(********************* G.D S.p.A. - Technical Department ***********************************
This program has been generated automatically from Application Designer DE&F
********************************************************************************************)
PROGRAM dbg_csp_case_transport_os_minorplow
VAR
  bwd_di_shd : digital_input_shadow;
  fwd_di_shd : digital_input_shadow;
  shift_do_shd : digital_output_shadow;
  shift_sact_shd : digital_actuator_shadow;
END_VAR

_objects_manager();

IF	g_application_status <> APPLICATION_STATUS_RUNNING
THEN
	RETURN;
END_IF

CASE process_get_mode(CONVERSION_this := dbg_root.prc) OF
	MODE_ABSENT,
	MODE_INACTIVE:
		RETURN;
	MODE_TEST:
		RETURN;
END_CASE

ACTION _objects_manager:
IF	objects_initialization()
THEN
	digital_input_shadow_init(
		sim_mode:= SHADOW_SIMULATION_MODE_AUTOMATIC, 
		father:= csp_case_transport_os_minorplow.bwd_di, 
		process:= dbg_root.prc, 
		CONVERSION_this:= bwd_di_shd);

	digital_input_shadow_init(
		sim_mode:= SHADOW_SIMULATION_MODE_AUTOMATIC, 
		father:= csp_case_transport_os_minorplow.fwd_di, 
		process:= dbg_root.prc, 
		CONVERSION_this:= fwd_di_shd);

	digital_output_shadow_init(
		sim_mode:= SHADOW_SIMULATION_MODE_AUTOMATIC, 
		father:= csp_case_transport_os_minorplow.shift_do, 
		process:= dbg_root.prc, 
		CONVERSION_this:= shift_do_shd);

	digital_actuator_shadow_init(
		sim_mode:= SHADOW_SIMULATION_MODE_AUTOMATIC, 
		father:= csp_case_transport_os_minorplow.shift_sact, 
		process:= dbg_root.prc, 
		CONVERSION_this:= shift_sact_shd);

	RETURN;
END_IF

IF	objects_running()
THEN
	digital_input_shadow_cycle(bwd_di_shd);
	digital_input_shadow_cycle(fwd_di_shd);
	digital_output_shadow_cycle(shift_do_shd);
	digital_actuator_shadow_cycle(shift_sact_shd);
END_IF
END_ACTION

END_PROGRAM

// ---- _Debug/dbg_csp_case_transport_os_trailing.TcPOU

(********************* G.D S.p.A. - Technical Department ***********************************
This program has been generated automatically from Application Designer DE&F
********************************************************************************************)
PROGRAM dbg_csp_case_transport_os_trailing
VAR
  axis_shd : axis_shadow;
END_VAR

_objects_manager();

IF	g_application_status <> APPLICATION_STATUS_RUNNING
THEN
	RETURN;
END_IF

CASE process_get_mode(CONVERSION_this := dbg_root.prc) OF
	MODE_ABSENT,
	MODE_INACTIVE:
		RETURN;
	MODE_TEST:
		RETURN;
END_CASE

ACTION _objects_manager:
IF	objects_initialization()
THEN
	axis_shadow_init(
		sim_mode:= SHADOW_SIMULATION_MODE_AUTOMATIC, 
		father:= csp_case_transport_os_trailing.axis, 
		process:= dbg_root.prc, 
		CONVERSION_this:= axis_shd);

	RETURN;
END_IF

IF	objects_running()
THEN
	axis_shadow_cycle(axis_shd);
END_IF
END_ACTION

END_PROGRAM

// ---- _Debug/dbg_csp_case_transport_tensioner.TcPOU

(********************* G.D S.p.A. - Technical Department ***********************************
This program has been generated automatically from Application Designer DE&F
********************************************************************************************)
PROGRAM dbg_csp_case_transport_tensioner
VAR
  chain_tensioner_do_shd : digital_output_shadow;
  chain_tensioner_sact_shd : digital_actuator_shadow;
END_VAR

_objects_manager();

IF	g_application_status <> APPLICATION_STATUS_RUNNING
THEN
	RETURN;
END_IF

CASE process_get_mode(CONVERSION_this := dbg_root.prc) OF
	MODE_ABSENT,
	MODE_INACTIVE:
		RETURN;
	MODE_TEST:
		RETURN;
END_CASE

ACTION _objects_manager:
IF	objects_initialization()
THEN
	digital_output_shadow_init(
		sim_mode:= SHADOW_SIMULATION_MODE_AUTOMATIC, 
		father:= csp_case_transport_tensioner.chain_tensioner_do, 
		process:= dbg_root.prc, 
		CONVERSION_this:= chain_tensioner_do_shd);

	digital_actuator_shadow_init(
		sim_mode:= SHADOW_SIMULATION_MODE_AUTOMATIC, 
		father:= csp_case_transport_tensioner.chain_tensioner_sact, 
		process:= dbg_root.prc, 
		CONVERSION_this:= chain_tensioner_sact_shd);

	RETURN;
END_IF

IF	objects_running()
THEN
	digital_output_shadow_cycle(chain_tensioner_do_shd);
	digital_actuator_shadow_cycle(chain_tensioner_sact_shd);
END_IF
END_ACTION

END_PROGRAM

// ---- _Debug/dbg_csp_case_transport_virtualmaster.TcPOU

(********************* G.D S.p.A. - Technical Department ***********************************
This program has been generated automatically from Application Designer DE&F
********************************************************************************************)
PROGRAM dbg_csp_case_transport_virtualmaster
VAR
  axis_shd : axis_shadow;
END_VAR

_objects_manager();

IF	g_application_status <> APPLICATION_STATUS_RUNNING
THEN
	RETURN;
END_IF

CASE process_get_mode(CONVERSION_this := dbg_root.prc) OF
	MODE_ABSENT,
	MODE_INACTIVE:
		RETURN;
	MODE_TEST:
		RETURN;
END_CASE

ACTION _objects_manager:
IF	objects_initialization()
THEN
	axis_shadow_init(
		sim_mode:= SHADOW_SIMULATION_MODE_AUTOMATIC, 
		father:= csp_case_transport_virtualmaster.axis, 
		process:= dbg_root.prc, 
		CONVERSION_this:= axis_shd);

	RETURN;
END_IF

IF	objects_running()
THEN
	axis_shadow_cycle(axis_shd);
END_IF
END_ACTION

END_PROGRAM

// ---- _Debug/dbg_csp_case_tr_accu_depth.TcPOU

(********************* G.D S.p.A. - Technical Department ***********************************
This program has been generated automatically from Application Designer DE&F
********************************************************************************************)
PROGRAM dbg_csp_case_tr_accu_depth
VAR
  axis_shd : axis_shadow;
END_VAR

_objects_manager();

IF	g_application_status <> APPLICATION_STATUS_RUNNING
THEN
	RETURN;
END_IF

CASE process_get_mode(CONVERSION_this := dbg_root.prc) OF
	MODE_ABSENT,
	MODE_INACTIVE:
		RETURN;
	MODE_TEST:
		RETURN;
END_CASE

ACTION _objects_manager:
IF	objects_initialization()
THEN
	axis_shadow_init(
		sim_mode:= SHADOW_SIMULATION_MODE_AUTOMATIC, 
		father:= csp_case_tr_accu_depth.axis, 
		process:= dbg_root.prc, 
		CONVERSION_this:= axis_shd);

	RETURN;
END_IF

IF	objects_running()
THEN
	axis_shadow_cycle(axis_shd);
END_IF
END_ACTION

END_PROGRAM

// ---- _Debug/dbg_csp_case_tr_accu_ls_width.TcPOU

(********************* G.D S.p.A. - Technical Department ***********************************
This program has been generated automatically from Application Designer DE&F
********************************************************************************************)
PROGRAM dbg_csp_case_tr_accu_ls_width
VAR
  axis_shd : axis_shadow;
END_VAR

_objects_manager();

IF	g_application_status <> APPLICATION_STATUS_RUNNING
THEN
	RETURN;
END_IF

CASE process_get_mode(CONVERSION_this := dbg_root.prc) OF
	MODE_ABSENT,
	MODE_INACTIVE:
		RETURN;
	MODE_TEST:
		RETURN;
END_CASE

ACTION _objects_manager:
IF	objects_initialization()
THEN
	axis_shadow_init(
		sim_mode:= SHADOW_SIMULATION_MODE_AUTOMATIC, 
		father:= csp_case_tr_accu_ls_width.axis, 
		process:= dbg_root.prc, 
		CONVERSION_this:= axis_shd);

	RETURN;
END_IF

IF	objects_running()
THEN
	axis_shadow_cycle(axis_shd);
END_IF
END_ACTION

END_PROGRAM

// ---- _Debug/dbg_csp_case_tr_accu_os_width.TcPOU

(********************* G.D S.p.A. - Technical Department ***********************************
This program has been generated automatically from Application Designer DE&F
********************************************************************************************)
PROGRAM dbg_csp_case_tr_accu_os_width
VAR
  axis_shd : axis_shadow;
END_VAR

_objects_manager();

IF	g_application_status <> APPLICATION_STATUS_RUNNING
THEN
	RETURN;
END_IF

CASE process_get_mode(CONVERSION_this := dbg_root.prc) OF
	MODE_ABSENT,
	MODE_INACTIVE:
		RETURN;
	MODE_TEST:
		RETURN;
END_CASE

ACTION _objects_manager:
IF	objects_initialization()
THEN
	axis_shadow_init(
		sim_mode:= SHADOW_SIMULATION_MODE_AUTOMATIC, 
		father:= csp_case_tr_accu_os_width.axis, 
		process:= dbg_root.prc, 
		CONVERSION_this:= axis_shd);

	RETURN;
END_IF

IF	objects_running()
THEN
	axis_shadow_cycle(axis_shd);
END_IF
END_ACTION

END_PROGRAM

// ---- _Debug/dbg_csp_case_tr_squaring_ls_leading.TcPOU

(********************* G.D S.p.A. - Technical Department ***********************************
This program has been generated automatically from Application Designer DE&F
********************************************************************************************)
PROGRAM dbg_csp_case_tr_squaring_ls_leading
VAR
  axis_shd : axis_shadow;
END_VAR

_objects_manager();

IF	g_application_status <> APPLICATION_STATUS_RUNNING
THEN
	RETURN;
END_IF

CASE process_get_mode(CONVERSION_this := dbg_root.prc) OF
	MODE_ABSENT,
	MODE_INACTIVE:
		RETURN;
	MODE_TEST:
		RETURN;
END_CASE

ACTION _objects_manager:
IF	objects_initialization()
THEN
	axis_shadow_init(
		sim_mode:= SHADOW_SIMULATION_MODE_AUTOMATIC, 
		father:= csp_case_tr_squaring_ls_leading.axis, 
		process:= dbg_root.prc, 
		CONVERSION_this:= axis_shd);

	RETURN;
END_IF

IF	objects_running()
THEN
	axis_shadow_cycle(axis_shd);
END_IF
END_ACTION

END_PROGRAM

// ---- _Debug/dbg_csp_case_tr_squaring_ls_trailing.TcPOU

(********************* G.D S.p.A. - Technical Department ***********************************
This program has been generated automatically from Application Designer DE&F
********************************************************************************************)
PROGRAM dbg_csp_case_tr_squaring_ls_trailing
VAR
  axis_shd : axis_shadow;
END_VAR

_objects_manager();

IF	g_application_status <> APPLICATION_STATUS_RUNNING
THEN
	RETURN;
END_IF

CASE process_get_mode(CONVERSION_this := dbg_root.prc) OF
	MODE_ABSENT,
	MODE_INACTIVE:
		RETURN;
	MODE_TEST:
		RETURN;
END_CASE

ACTION _objects_manager:
IF	objects_initialization()
THEN
	axis_shadow_init(
		sim_mode:= SHADOW_SIMULATION_MODE_AUTOMATIC, 
		father:= csp_case_tr_squaring_ls_trailing.axis, 
		process:= dbg_root.prc, 
		CONVERSION_this:= axis_shd);

	RETURN;
END_IF

IF	objects_running()
THEN
	axis_shadow_cycle(axis_shd);
END_IF
END_ACTION

END_PROGRAM

// ---- _Debug/dbg_csp_case_tr_squaring_os_leading.TcPOU

(********************* G.D S.p.A. - Technical Department ***********************************
This program has been generated automatically from Application Designer DE&F
********************************************************************************************)
PROGRAM dbg_csp_case_tr_squaring_os_leading
VAR
  axis_shd : axis_shadow;
END_VAR

_objects_manager();

IF	g_application_status <> APPLICATION_STATUS_RUNNING
THEN
	RETURN;
END_IF

CASE process_get_mode(CONVERSION_this := dbg_root.prc) OF
	MODE_ABSENT,
	MODE_INACTIVE:
		RETURN;
	MODE_TEST:
		RETURN;
END_CASE

ACTION _objects_manager:
IF	objects_initialization()
THEN
	axis_shadow_init(
		sim_mode:= SHADOW_SIMULATION_MODE_AUTOMATIC, 
		father:= csp_case_tr_squaring_os_leading.axis, 
		process:= dbg_root.prc, 
		CONVERSION_this:= axis_shd);

	RETURN;
END_IF

IF	objects_running()
THEN
	axis_shadow_cycle(axis_shd);
END_IF
END_ACTION

END_PROGRAM

// ---- _Debug/dbg_csp_case_tr_squaring_os_trailing.TcPOU

(********************* G.D S.p.A. - Technical Department ***********************************
This program has been generated automatically from Application Designer DE&F
********************************************************************************************)
PROGRAM dbg_csp_case_tr_squaring_os_trailing
VAR
  axis_shd : axis_shadow;
END_VAR

_objects_manager();

IF	g_application_status <> APPLICATION_STATUS_RUNNING
THEN
	RETURN;
END_IF

CASE process_get_mode(CONVERSION_this := dbg_root.prc) OF
	MODE_ABSENT,
	MODE_INACTIVE:
		RETURN;
	MODE_TEST:
		RETURN;
END_CASE

ACTION _objects_manager:
IF	objects_initialization()
THEN
	axis_shadow_init(
		sim_mode:= SHADOW_SIMULATION_MODE_AUTOMATIC, 
		father:= csp_case_tr_squaring_os_trailing.axis, 
		process:= dbg_root.prc, 
		CONVERSION_this:= axis_shd);

	RETURN;
END_IF

IF	objects_running()
THEN
	axis_shadow_cycle(axis_shd);
END_IF
END_ACTION

END_PROGRAM

// ---- _Debug/dbg_csp_case_virtualmaster.TcPOU

(********************* G.D S.p.A. - Technical Department ***********************************
This program has been generated automatically from Application Designer DE&F
********************************************************************************************)
PROGRAM dbg_csp_case_virtualmaster
VAR
  axis_shd : axis_shadow;
END_VAR

_objects_manager();

IF	g_application_status <> APPLICATION_STATUS_RUNNING
THEN
	RETURN;
END_IF

CASE process_get_mode(CONVERSION_this := dbg_root.prc) OF
	MODE_ABSENT,
	MODE_INACTIVE:
		RETURN;
	MODE_TEST:
		RETURN;
END_CASE

ACTION _objects_manager:
IF	objects_initialization()
THEN
	axis_shadow_init(
		sim_mode:= SHADOW_SIMULATION_MODE_AUTOMATIC, 
		father:= csp_case_virtualmaster.axis, 
		process:= dbg_root.prc, 
		CONVERSION_this:= axis_shd);

	RETURN;
END_IF

IF	objects_running()
THEN
	axis_shadow_cycle(axis_shd);
END_IF
END_ACTION

END_PROGRAM

// ---- _Debug/dbg_csp_main_jogmanager.TcPOU

(********************* G.D S.p.A. - Technical Department ***********************************
This program has been generated automatically from Application Designer DE&F
********************************************************************************************)
PROGRAM dbg_csp_main_jogmanager
VAR
  di_pendant_negative_shd : digital_input_shadow;
  di_pendant_positive_shd : digital_input_shadow;
END_VAR

_objects_manager();

IF	g_application_status <> APPLICATION_STATUS_RUNNING
THEN
	RETURN;
END_IF

CASE process_get_mode(CONVERSION_this := dbg_root.prc) OF
	MODE_ABSENT,
	MODE_INACTIVE:
		RETURN;
	MODE_TEST:
		RETURN;
END_CASE

ACTION _objects_manager:
IF	objects_initialization()
THEN
	digital_input_shadow_init(
		sim_mode:= SHADOW_SIMULATION_MODE_AUTOMATIC, 
		father:= csp_main_jogmanager.di_pendant_negative, 
		process:= dbg_root.prc, 
		CONVERSION_this:= di_pendant_negative_shd);

	digital_input_shadow_init(
		sim_mode:= SHADOW_SIMULATION_MODE_AUTOMATIC, 
		father:= csp_main_jogmanager.di_pendant_positive, 
		process:= dbg_root.prc, 
		CONVERSION_this:= di_pendant_positive_shd);

	RETURN;
END_IF

IF	objects_running()
THEN
	digital_input_shadow_cycle(di_pendant_negative_shd);
	digital_input_shadow_cycle(di_pendant_positive_shd);
END_IF
END_ACTION

END_PROGRAM

// ---- _Debug/dbg_csp_main_motorization_virtualmanager.TcPOU

(********************* G.D S.p.A. - Technical Department ***********************************
This program has been generated automatically from Application Designer DE&F
********************************************************************************************)
PROGRAM dbg_csp_main_motorization_virtualmanager
VAR
  axis_shd : axis_shadow;
  machine_periodicity_axis_shd : axis_shadow;
  virtual_master_test_shd : axis_shadow;
END_VAR

_objects_manager();

IF	g_application_status <> APPLICATION_STATUS_RUNNING
THEN
	RETURN;
END_IF

CASE process_get_mode(CONVERSION_this := dbg_root.prc) OF
	MODE_ABSENT,
	MODE_INACTIVE:
		RETURN;
	MODE_TEST:
		RETURN;
END_CASE

ACTION _objects_manager:
IF	objects_initialization()
THEN
	axis_shadow_init(
		sim_mode:= SHADOW_SIMULATION_MODE_AUTOMATIC, 
		father:= csp_main_motorization_virtualmanager.axis, 
		process:= dbg_root.prc, 
		CONVERSION_this:= axis_shd);

	axis_shadow_init(
		sim_mode:= SHADOW_SIMULATION_MODE_AUTOMATIC, 
		father:= csp_main_motorization_virtualmanager.machine_periodicity_axis, 
		process:= dbg_root.prc, 
		CONVERSION_this:= machine_periodicity_axis_shd);

	axis_shadow_init(
		sim_mode:= SHADOW_SIMULATION_MODE_AUTOMATIC, 
		father:= csp_main_motorization_virtualmanager.virtual_master_test, 
		process:= dbg_root.prc, 
		CONVERSION_this:= virtual_master_test_shd);

	RETURN;
END_IF

IF	objects_running()
THEN
	axis_shadow_cycle(axis_shd);
	axis_shadow_cycle(machine_periodicity_axis_shd);
	axis_shadow_cycle(virtual_master_test_shd);
END_IF
END_ACTION

END_PROGRAM

// ---- _Debug/dbg_csp_main_services.TcPOU

(********************* G.D S.p.A. - Technical Department ***********************************
This program has been generated automatically from Application Designer DE&F
********************************************************************************************)
PROGRAM dbg_csp_main_services
VAR
  reset_output_test_shd : digital_output_shadow;
END_VAR

_objects_manager();

IF	g_application_status <> APPLICATION_STATUS_RUNNING
THEN
	RETURN;
END_IF

CASE process_get_mode(CONVERSION_this := dbg_root.prc) OF
	MODE_ABSENT,
	MODE_INACTIVE:
		RETURN;
	MODE_TEST:
		RETURN;
END_CASE

ACTION _objects_manager:
IF	objects_initialization()
THEN
	digital_output_shadow_init(
		sim_mode:= SHADOW_SIMULATION_MODE_AUTOMATIC, 
		father:= csp_main_services.reset_output_test, 
		process:= dbg_root.prc, 
		CONVERSION_this:= reset_output_test_shd);

	RETURN;
END_IF

IF	objects_running()
THEN
	digital_output_shadow_cycle(reset_output_test_shd);
END_IF
END_ACTION

END_PROGRAM

// ---- _Debug/dbg_csp_transfer_accumulator_accu_convdepth.TcPOU

(********************* G.D S.p.A. - Technical Department ***********************************
This program has been generated automatically from Application Designer DE&F
********************************************************************************************)
PROGRAM dbg_csp_transfer_accumulator_accu_convdepth
VAR
  axis_shd : axis_shadow;
END_VAR

_objects_manager();

IF	g_application_status <> APPLICATION_STATUS_RUNNING
THEN
	RETURN;
END_IF

CASE process_get_mode(CONVERSION_this := dbg_root.prc) OF
	MODE_ABSENT,
	MODE_INACTIVE:
		RETURN;
	MODE_TEST:
		RETURN;
END_CASE

ACTION _objects_manager:
IF	objects_initialization()
THEN
	axis_shadow_init(
		sim_mode:= SHADOW_SIMULATION_MODE_AUTOMATIC, 
		father:= csp_transfer_accumulator_accu_convdepth.axis, 
		process:= dbg_root.prc, 
		CONVERSION_this:= axis_shd);

	RETURN;
END_IF

IF	objects_running()
THEN
	axis_shadow_cycle(axis_shd);
END_IF
END_ACTION

END_PROGRAM

// ---- _Debug/dbg_csp_transfer_accumulator_accu_depth.TcPOU

(********************* G.D S.p.A. - Technical Department ***********************************
This program has been generated automatically from Application Designer DE&F
********************************************************************************************)
PROGRAM dbg_csp_transfer_accumulator_accu_depth
VAR
  axis_shd : axis_shadow;
END_VAR

_objects_manager();

IF	g_application_status <> APPLICATION_STATUS_RUNNING
THEN
	RETURN;
END_IF

CASE process_get_mode(CONVERSION_this := dbg_root.prc) OF
	MODE_ABSENT,
	MODE_INACTIVE:
		RETURN;
	MODE_TEST:
		RETURN;
END_CASE

ACTION _objects_manager:
IF	objects_initialization()
THEN
	axis_shadow_init(
		sim_mode:= SHADOW_SIMULATION_MODE_AUTOMATIC, 
		father:= csp_transfer_accumulator_accu_depth.axis, 
		process:= dbg_root.prc, 
		CONVERSION_this:= axis_shd);

	RETURN;
END_IF

IF	objects_running()
THEN
	axis_shadow_cycle(axis_shd);
END_IF
END_ACTION

END_PROGRAM

// ---- _Debug/dbg_csp_transfer_accumulator_accu_topraillength.TcPOU

(********************* G.D S.p.A. - Technical Department ***********************************
This program has been generated automatically from Application Designer DE&F
********************************************************************************************)
PROGRAM dbg_csp_transfer_accumulator_accu_topraillength
VAR
  axis_shd : axis_shadow;
END_VAR

_objects_manager();

IF	g_application_status <> APPLICATION_STATUS_RUNNING
THEN
	RETURN;
END_IF

CASE process_get_mode(CONVERSION_this := dbg_root.prc) OF
	MODE_ABSENT,
	MODE_INACTIVE:
		RETURN;
	MODE_TEST:
		RETURN;
END_CASE

ACTION _objects_manager:
(*IF	objects_initialization()
THEN
	axis_shadow_init(
		sim_mode:= SHADOW_SIMULATION_MODE_AUTOMATIC, 
		father:= csp_transfer_accumulator_accu_topraillength.axis, 
		process:= dbg_root.prc, 
		CONVERSION_this:= axis_shd);

	RETURN;
END_IF

IF	objects_running()
THEN
	axis_shadow_cycle(axis_shd);
END_IF
*)
END_ACTION

END_PROGRAM

// ---- _Debug/dbg_csp_transfer_accumulator_accu_toprailwidth.TcPOU

(********************* G.D S.p.A. - Technical Department ***********************************
This program has been generated automatically from Application Designer DE&F
********************************************************************************************)
PROGRAM dbg_csp_transfer_accumulator_accu_toprailwidth
VAR
  axis_shd : axis_shadow;
END_VAR

_objects_manager();

IF	g_application_status <> APPLICATION_STATUS_RUNNING
THEN
	RETURN;
END_IF

CASE process_get_mode(CONVERSION_this := dbg_root.prc) OF
	MODE_ABSENT,
	MODE_INACTIVE:
		RETURN;
	MODE_TEST:
		RETURN;
END_CASE

ACTION _objects_manager:
(*IF	objects_initialization()
THEN
	axis_shadow_init(
		sim_mode:= SHADOW_SIMULATION_MODE_AUTOMATIC, 
		father:= csp_transfer_accumulator_accu_toprailwidth.axis, 
		process:= dbg_root.prc, 
		CONVERSION_this:= axis_shd);

	RETURN;
END_IF

IF	objects_running()
THEN
	axis_shadow_cycle(axis_shd);
END_IF*)
END_ACTION

END_PROGRAM

// ---- _Debug/dbg_csp_transfer_accumulator_belt.TcPOU

(********************* G.D S.p.A. - Technical Department ***********************************
This program has been generated automatically from Application Designer DE&F
********************************************************************************************)
PROGRAM dbg_csp_transfer_accumulator_belt
VAR
  axis_shd : axis_shadow;
END_VAR

_objects_manager();

IF	g_application_status <> APPLICATION_STATUS_RUNNING
THEN
	RETURN;
END_IF

CASE process_get_mode(CONVERSION_this := dbg_root.prc) OF
	MODE_ABSENT,
	MODE_INACTIVE:
		RETURN;
	MODE_TEST:
		RETURN;
END_CASE

ACTION _objects_manager:
IF	objects_initialization()
THEN
	axis_shadow_init(
		sim_mode:= SHADOW_SIMULATION_MODE_AUTOMATIC, 
		father:= csp_transfer_accumulator_belt.axis, 
		process:= dbg_root.prc, 
		CONVERSION_this:= axis_shd);

	RETURN;
END_IF

IF	objects_running()
THEN
	axis_shadow_cycle(axis_shd);
END_IF
END_ACTION

END_PROGRAM

// ---- _Debug/dbg_csp_transfer_accumulator_finger_ls.TcPOU

(********************* G.D S.p.A. - Technical Department ***********************************
This program has been generated automatically from Application Designer DE&F
********************************************************************************************)
PROGRAM dbg_csp_transfer_accumulator_finger_ls
VAR
  axis_shd : axis_shadow;
END_VAR

_objects_manager();

IF	g_application_status <> APPLICATION_STATUS_RUNNING
THEN
	RETURN;
END_IF

CASE process_get_mode(CONVERSION_this := dbg_root.prc) OF
	MODE_ABSENT,
	MODE_INACTIVE:
		RETURN;
	MODE_TEST:
		RETURN;
END_CASE

ACTION _objects_manager:
IF	objects_initialization()
THEN
	axis_shadow_init(
		sim_mode:= SHADOW_SIMULATION_MODE_AUTOMATIC, 
		father:= csp_transfer_accumulator_finger_ls.axis, 
		process:= dbg_root.prc, 
		CONVERSION_this:= axis_shd);

	RETURN;
END_IF

IF	objects_running()
THEN
	axis_shadow_cycle(axis_shd);
END_IF
END_ACTION

END_PROGRAM

// ---- _Debug/dbg_csp_transfer_accumulator_finger_os.TcPOU

(********************* G.D S.p.A. - Technical Department ***********************************
This program has been generated automatically from Application Designer DE&F
********************************************************************************************)
PROGRAM dbg_csp_transfer_accumulator_finger_os
VAR
  axis_shd : axis_shadow;
END_VAR

_objects_manager();

IF	g_application_status <> APPLICATION_STATUS_RUNNING
THEN
	RETURN;
END_IF

CASE process_get_mode(CONVERSION_this := dbg_root.prc) OF
	MODE_ABSENT,
	MODE_INACTIVE:
		RETURN;
	MODE_TEST:
		RETURN;
END_CASE

ACTION _objects_manager:
IF	objects_initialization()
THEN
	axis_shadow_init(
		sim_mode:= SHADOW_SIMULATION_MODE_AUTOMATIC, 
		father:= csp_transfer_accumulator_finger_os.axis, 
		process:= dbg_root.prc, 
		CONVERSION_this:= axis_shd);

	RETURN;
END_IF

IF	objects_running()
THEN
	axis_shadow_cycle(axis_shd);
END_IF
END_ACTION

END_PROGRAM

// ---- _Debug/dbg_csp_transfer_accumulator_lift.TcPOU

(********************* G.D S.p.A. - Technical Department ***********************************
This program has been generated automatically from Application Designer DE&F
********************************************************************************************)
PROGRAM dbg_csp_transfer_accumulator_lift
VAR
  axis_shd : axis_shadow;
END_VAR

_objects_manager();

IF	g_application_status <> APPLICATION_STATUS_RUNNING
THEN
	RETURN;
END_IF

CASE process_get_mode(CONVERSION_this := dbg_root.prc) OF
	MODE_ABSENT,
	MODE_INACTIVE:
		RETURN;
	MODE_TEST:
		RETURN;
END_CASE

ACTION _objects_manager:
IF	objects_initialization()
THEN
	axis_shadow_init(
		sim_mode:= SHADOW_SIMULATION_MODE_AUTOMATIC, 
		father:= csp_transfer_accumulator_lift.axis, 
		process:= dbg_root.prc, 
		CONVERSION_this:= axis_shd);

	RETURN;
END_IF

IF	objects_running()
THEN
	axis_shadow_cycle(axis_shd);
END_IF
END_ACTION

END_PROGRAM

// ---- _Debug/dbg_csp_transfer_accumulator_virtualmaster.TcPOU

(********************* G.D S.p.A. - Technical Department ***********************************
This program has been generated automatically from Application Designer DE&F
********************************************************************************************)
PROGRAM dbg_csp_transfer_accumulator_virtualmaster
VAR
  axis_shd : axis_shadow;
END_VAR

_objects_manager();

IF	g_application_status <> APPLICATION_STATUS_RUNNING
THEN
	RETURN;
END_IF

CASE process_get_mode(CONVERSION_this := dbg_root.prc) OF
	MODE_ABSENT,
	MODE_INACTIVE:
		RETURN;
	MODE_TEST:
		RETURN;
END_CASE

ACTION _objects_manager:
IF	objects_initialization()
THEN
	axis_shadow_init(
		sim_mode:= SHADOW_SIMULATION_MODE_AUTOMATIC, 
		father:= csp_transfer_accumulator_virtualmaster.axis, 
		process:= dbg_root.prc, 
		CONVERSION_this:= axis_shd);

	RETURN;
END_IF

IF	objects_running()
THEN
	axis_shadow_cycle(axis_shd);
END_IF
END_ACTION

END_PROGRAM

// ---- _Debug/dbg_csp_transfer_crosspusher_follower.TcPOU

(********************* G.D S.p.A. - Technical Department ***********************************
This program has been generated automatically from Application Designer DE&F
********************************************************************************************)
PROGRAM dbg_csp_transfer_crosspusher_follower
VAR
  axis_shd : axis_shadow;
END_VAR

_objects_manager();

IF	g_application_status <> APPLICATION_STATUS_RUNNING
THEN
	RETURN;
END_IF

CASE process_get_mode(CONVERSION_this := dbg_root.prc) OF
	MODE_ABSENT,
	MODE_INACTIVE:
		RETURN;
	MODE_TEST:
		RETURN;
END_CASE

ACTION _objects_manager:
IF	objects_initialization()
THEN
	axis_shadow_init(
		sim_mode:= SHADOW_SIMULATION_MODE_AUTOMATIC, 
		father:= csp_transfer_crosspusher_follower.axis, 
		process:= dbg_root.prc, 
		CONVERSION_this:= axis_shd);

	RETURN;
END_IF

IF	objects_running()
THEN
	axis_shadow_cycle(axis_shd);
END_IF
END_ACTION

END_PROGRAM

// ---- _Debug/dbg_csp_transfer_crosspusher_horizontal.TcPOU

(********************* G.D S.p.A. - Technical Department ***********************************
This program has been generated automatically from Application Designer DE&F
********************************************************************************************)
PROGRAM dbg_csp_transfer_crosspusher_horizontal
VAR
  axis_shd : axis_shadow;
END_VAR

_objects_manager();

IF	g_application_status <> APPLICATION_STATUS_RUNNING
THEN
	RETURN;
END_IF

CASE process_get_mode(CONVERSION_this := dbg_root.prc) OF
	MODE_ABSENT,
	MODE_INACTIVE:
		RETURN;
	MODE_TEST:
		RETURN;
END_CASE

ACTION _objects_manager:
IF	objects_initialization()
THEN
	axis_shadow_init(
		sim_mode:= SHADOW_SIMULATION_MODE_AUTOMATIC, 
		father:= csp_transfer_crosspusher_horizontal.axis, 
		process:= dbg_root.prc, 
		CONVERSION_this:= axis_shd);

	RETURN;
END_IF

IF	objects_running()
THEN
	axis_shadow_cycle(axis_shd);
END_IF
END_ACTION

END_PROGRAM

// ---- _Debug/dbg_csp_transfer_crosspusher_reject.TcPOU

(********************* G.D S.p.A. - Technical Department ***********************************
This program has been generated automatically from Application Designer DE&F
********************************************************************************************)
PROGRAM dbg_csp_transfer_crosspusher_reject
VAR
  backup_di_shd : digital_input_shadow;
  backup_di_dchk_shd : digital_check_shadow;
  extend_do_shd : digital_output_shadow;
  present_di_shd : digital_input_shadow;
  reject_present_check_shd : digital_check_shadow;
  retracted_di_shd : digital_input_shadow;
END_VAR

_objects_manager();

IF	g_application_status <> APPLICATION_STATUS_RUNNING
THEN
	RETURN;
END_IF

CASE process_get_mode(CONVERSION_this := dbg_root.prc) OF
	MODE_ABSENT,
	MODE_INACTIVE:
		RETURN;
	MODE_TEST:
		RETURN;
END_CASE

ACTION _objects_manager:
IF	objects_initialization()
THEN
	digital_input_shadow_init(
		sim_mode:= SHADOW_SIMULATION_MODE_AUTOMATIC, 
		father:= csp_transfer_crosspusher_reject.backup_di, 
		process:= dbg_root.prc, 
		CONVERSION_this:= backup_di_shd);

	digital_check_shadow_init(
		sim_mode:= SHADOW_SIMULATION_MODE_AUTOMATIC, 
		father:= csp_transfer_crosspusher_reject.backup_di_dchk, 
		process:= dbg_root.prc, 
		CONVERSION_this:= backup_di_dchk_shd);

	digital_output_shadow_init(
		sim_mode:= SHADOW_SIMULATION_MODE_AUTOMATIC, 
		father:= csp_transfer_crosspusher_reject.extend_do, 
		process:= dbg_root.prc, 
		CONVERSION_this:= extend_do_shd);

	digital_input_shadow_init(
		sim_mode:= SHADOW_SIMULATION_MODE_AUTOMATIC, 
		father:= csp_transfer_crosspusher_reject.present_di, 
		process:= dbg_root.prc, 
		CONVERSION_this:= present_di_shd);

	digital_check_shadow_init(
		sim_mode:= SHADOW_SIMULATION_MODE_AUTOMATIC, 
		father:= csp_transfer_crosspusher_reject.reject_present_check, 
		process:= dbg_root.prc, 
		CONVERSION_this:= reject_present_check_shd);

	digital_input_shadow_init(
		sim_mode:= SHADOW_SIMULATION_MODE_AUTOMATIC, 
		father:= csp_transfer_crosspusher_reject.retracted_di, 
		process:= dbg_root.prc, 
		CONVERSION_this:= retracted_di_shd);

	RETURN;
END_IF

IF	objects_running()
THEN
	digital_input_shadow_cycle(backup_di_shd);
	digital_check_shadow_cycle(backup_di_dchk_shd);
	digital_output_shadow_cycle(extend_do_shd);
	digital_input_shadow_cycle(present_di_shd);
	digital_check_shadow_cycle(reject_present_check_shd);
	digital_input_shadow_cycle(retracted_di_shd);
END_IF
END_ACTION

END_PROGRAM

// ---- _Debug/dbg_csp_transfer_crosspusher_sensors.TcPOU

(********************* G.D S.p.A. - Technical Department ***********************************
This program has been generated automatically from Application Designer DE&F
********************************************************************************************)
PROGRAM dbg_csp_transfer_crosspusher_sensors
VAR
  high_achk_shd : analog_check_shadow;
  high_ai_shd : analog_input_shadow;
END_VAR

_objects_manager();

IF	g_application_status <> APPLICATION_STATUS_RUNNING
THEN
	RETURN;
END_IF

CASE process_get_mode(CONVERSION_this := dbg_root.prc) OF
	MODE_ABSENT,
	MODE_INACTIVE:
		RETURN;
	MODE_TEST:
		RETURN;
END_CASE

ACTION _objects_manager:
IF	objects_initialization()
THEN


	RETURN;
END_IF

IF	objects_running()
THEN
;
END_IF
END_ACTION

END_PROGRAM

// ---- _Debug/dbg_csp_transfer_crosspusher_vertical.TcPOU

(********************* G.D S.p.A. - Technical Department ***********************************
This program has been generated automatically from Application Designer DE&F
********************************************************************************************)
PROGRAM dbg_csp_transfer_crosspusher_vertical
VAR
  axis_shd : axis_shadow;
END_VAR

_objects_manager();

IF	g_application_status <> APPLICATION_STATUS_RUNNING
THEN
	RETURN;
END_IF

CASE process_get_mode(CONVERSION_this := dbg_root.prc) OF
	MODE_ABSENT,
	MODE_INACTIVE:
		RETURN;
	MODE_TEST:
		RETURN;
END_CASE

ACTION _objects_manager:
IF	objects_initialization()
THEN
	axis_shadow_init(
		sim_mode:= SHADOW_SIMULATION_MODE_AUTOMATIC, 
		father:= csp_transfer_crosspusher_vertical.axis, 
		process:= dbg_root.prc, 
		CONVERSION_this:= axis_shd);

	RETURN;
END_IF

IF	objects_running()
THEN
	axis_shadow_cycle(axis_shd);
END_IF
END_ACTION

END_PROGRAM

// ---- _Debug/dbg_csp_transfer_crosspusher_virtualmaster.TcPOU

(********************* G.D S.p.A. - Technical Department ***********************************
This program has been generated automatically from Application Designer DE&F
********************************************************************************************)
PROGRAM dbg_csp_transfer_crosspusher_virtualmaster
VAR
  axis_shd : axis_shadow;
END_VAR

_objects_manager();

IF	g_application_status <> APPLICATION_STATUS_RUNNING
THEN
	RETURN;
END_IF

CASE process_get_mode(CONVERSION_this := dbg_root.prc) OF
	MODE_ABSENT,
	MODE_INACTIVE:
		RETURN;
	MODE_TEST:
		RETURN;
END_CASE

ACTION _objects_manager:
IF	objects_initialization()
THEN
	axis_shadow_init(
		sim_mode:= SHADOW_SIMULATION_MODE_AUTOMATIC, 
		father:= csp_transfer_crosspusher_virtualmaster.axis, 
		process:= dbg_root.prc, 
		CONVERSION_this:= axis_shd);

	RETURN;
END_IF

IF	objects_running()
THEN
	axis_shadow_cycle(axis_shd);
END_IF
END_ACTION

END_PROGRAM

// ---- _Debug/dbg_csp_transfer_infeed.TcPOU

(********************* G.D S.p.A. - Technical Department ***********************************
This program has been generated automatically from Application Designer DE&F
********************************************************************************************)
PROGRAM dbg_csp_transfer_infeed
VAR
  run_do_shd : digital_output_shadow;
  running_di_shd : digital_input_shadow;
  speed_ao_shd : analog_output_shadow;
END_VAR

_objects_manager();

IF	g_application_status <> APPLICATION_STATUS_RUNNING
THEN
	RETURN;
END_IF

CASE process_get_mode(CONVERSION_this := dbg_root.prc) OF
	MODE_ABSENT,
	MODE_INACTIVE:
		RETURN;
	MODE_TEST:
		RETURN;
END_CASE

ACTION _objects_manager:
IF	objects_initialization()
THEN
	digital_output_shadow_init(
		sim_mode:= SHADOW_SIMULATION_MODE_AUTOMATIC, 
		father:= csp_transfer_infeed.run_do, 
		process:= dbg_root.prc, 
		CONVERSION_this:= run_do_shd);


	RETURN;
END_IF

IF	objects_running()
THEN
	digital_output_shadow_cycle(run_do_shd);
	digital_input_shadow_cycle(running_di_shd);
	analog_output_shadow_cycle(speed_ao_shd);
END_IF
END_ACTION

END_PROGRAM

// ---- _Debug/dbg_csp_transfer_infeed_accumulation_belt.TcPOU

(********************* G.D S.p.A. - Technical Department ***********************************
This program has been generated automatically from Application Designer DE&F
********************************************************************************************)
PROGRAM dbg_csp_transfer_infeed_accumulation_belt
VAR
  axis_shd : axis_shadow;
END_VAR

_objects_manager();

IF	g_application_status <> APPLICATION_STATUS_RUNNING
THEN
	RETURN;
END_IF

CASE process_get_mode(CONVERSION_this := dbg_root.prc) OF
	MODE_ABSENT,
	MODE_INACTIVE:
		RETURN;
	MODE_TEST:
		RETURN;
END_CASE

ACTION _objects_manager:
IF	objects_initialization()
THEN
	axis_shadow_init(
		sim_mode:= SHADOW_SIMULATION_MODE_AUTOMATIC, 
		father:= csp_transfer_infeed_accumulation_belt.axis, 
		process:= dbg_root.prc, 
		CONVERSION_this:= axis_shd);

	RETURN;
END_IF

IF	objects_running()
THEN
	axis_shadow_cycle(axis_shd);
END_IF
END_ACTION

END_PROGRAM

// ---- _Debug/dbg_csp_transfer_infeed_accumulation_level_low.TcPOU

(********************* G.D S.p.A. - Technical Department ***********************************
This program has been generated automatically from Application Designer DE&F
********************************************************************************************)
PROGRAM dbg_csp_transfer_infeed_accumulation_level_low
VAR
  di_shd : digital_input_shadow;
END_VAR

_objects_manager();

IF	g_application_status <> APPLICATION_STATUS_RUNNING
THEN
	RETURN;
END_IF

CASE process_get_mode(CONVERSION_this := dbg_root.prc) OF
	MODE_ABSENT,
	MODE_INACTIVE:
		RETURN;
	MODE_TEST:
		RETURN;
END_CASE

ACTION _objects_manager:
IF	objects_initialization()
THEN
	digital_input_shadow_init(
		sim_mode:= SHADOW_SIMULATION_MODE_AUTOMATIC, 
		father:= csp_transfer_infeed_accumulation_level_low.di, 
		process:= dbg_root.prc, 
		CONVERSION_this:= di_shd);

	RETURN;
END_IF

IF	objects_running()
THEN
	digital_input_shadow_cycle(di_shd);
END_IF
END_ACTION

END_PROGRAM

// ---- _Debug/dbg_csp_transfer_infeed_accumulation_level_max.TcPOU

(********************* G.D S.p.A. - Technical Department ***********************************
This program has been generated automatically from Application Designer DE&F
********************************************************************************************)
PROGRAM dbg_csp_transfer_infeed_accumulation_level_max
VAR
  di_shd : digital_input_shadow;
END_VAR

_objects_manager();

IF	g_application_status <> APPLICATION_STATUS_RUNNING
THEN
	RETURN;
END_IF

CASE process_get_mode(CONVERSION_this := dbg_root.prc) OF
	MODE_ABSENT,
	MODE_INACTIVE:
		RETURN;
	MODE_TEST:
		RETURN;
END_CASE

ACTION _objects_manager:
IF	objects_initialization()
THEN
	digital_input_shadow_init(
		sim_mode:= SHADOW_SIMULATION_MODE_AUTOMATIC, 
		father:= csp_transfer_infeed_accumulation_level_max.di, 
		process:= dbg_root.prc, 
		CONVERSION_this:= di_shd);

	RETURN;
END_IF

IF	objects_running()
THEN
	digital_input_shadow_cycle(di_shd);
END_IF
END_ACTION

END_PROGRAM

// ---- _Debug/dbg_csp_transfer_infeed_accumulation_level_min.TcPOU

(********************* G.D S.p.A. - Technical Department ***********************************
This program has been generated automatically from Application Designer DE&F
********************************************************************************************)
PROGRAM dbg_csp_transfer_infeed_accumulation_level_min
VAR
  di_shd : digital_input_shadow;
END_VAR

_objects_manager();

IF	g_application_status <> APPLICATION_STATUS_RUNNING
THEN
	RETURN;
END_IF

CASE process_get_mode(CONVERSION_this := dbg_root.prc) OF
	MODE_ABSENT,
	MODE_INACTIVE:
		RETURN;
	MODE_TEST:
		RETURN;
END_CASE

ACTION _objects_manager:
IF	objects_initialization()
THEN
	digital_input_shadow_init(
		sim_mode:= SHADOW_SIMULATION_MODE_AUTOMATIC, 
		father:= csp_transfer_infeed_accumulation_level_min.di, 
		process:= dbg_root.prc, 
		CONVERSION_this:= di_shd);

	RETURN;
END_IF

IF	objects_running()
THEN
	digital_input_shadow_cycle(di_shd);
END_IF
END_ACTION

END_PROGRAM

// ---- _Debug/dbg_csp_transfer_infeed_accumulation_level_normal.TcPOU

(********************* G.D S.p.A. - Technical Department ***********************************
This program has been generated automatically from Application Designer DE&F
********************************************************************************************)
PROGRAM dbg_csp_transfer_infeed_accumulation_level_normal
VAR
  di_shd : digital_input_shadow;
END_VAR

_objects_manager();

IF	g_application_status <> APPLICATION_STATUS_RUNNING
THEN
	RETURN;
END_IF

CASE process_get_mode(CONVERSION_this := dbg_root.prc) OF
	MODE_ABSENT,
	MODE_INACTIVE:
		RETURN;
	MODE_TEST:
		RETURN;
END_CASE

ACTION _objects_manager:
IF	objects_initialization()
THEN
	digital_input_shadow_init(
		sim_mode:= SHADOW_SIMULATION_MODE_AUTOMATIC, 
		father:= csp_transfer_infeed_accumulation_level_normal.di, 
		process:= dbg_root.prc, 
		CONVERSION_this:= di_shd);

	RETURN;
END_IF

IF	objects_running()
THEN
	digital_input_shadow_cycle(di_shd);
END_IF
END_ACTION

END_PROGRAM

// ---- _Debug/dbg_csp_transfer_infeed_accu_depth.TcPOU

(********************* G.D S.p.A. - Technical Department ***********************************
This program has been generated automatically from Application Designer DE&F
********************************************************************************************)
PROGRAM dbg_csp_transfer_infeed_accu_depth
VAR
  axis_shd : axis_shadow;
END_VAR

_objects_manager();

IF	g_application_status <> APPLICATION_STATUS_RUNNING
THEN
	RETURN;
END_IF

CASE process_get_mode(CONVERSION_this := dbg_root.prc) OF
	MODE_ABSENT,
	MODE_INACTIVE:
		RETURN;
	MODE_TEST:
		RETURN;
END_CASE

ACTION _objects_manager:
IF	objects_initialization()
THEN
	axis_shadow_init(
		sim_mode:= SHADOW_SIMULATION_MODE_AUTOMATIC, 
		father:= csp_transfer_infeed_accu_depth.axis, 
		process:= dbg_root.prc, 
		CONVERSION_this:= axis_shd);

	RETURN;
END_IF

IF	objects_running()
THEN
	axis_shadow_cycle(axis_shd);
END_IF
END_ACTION

END_PROGRAM

// ---- _Debug/dbg_csp_transfer_infeed_accu_waterfalladjust.TcPOU

(********************* G.D S.p.A. - Technical Department ***********************************
This program has been generated automatically from Application Designer DE&F
********************************************************************************************)
PROGRAM dbg_csp_transfer_infeed_accu_waterfalladjust
VAR
  axis_shd : axis_shadow;
END_VAR

_objects_manager();

IF	g_application_status <> APPLICATION_STATUS_RUNNING
THEN
	RETURN;
END_IF

CASE process_get_mode(CONVERSION_this := dbg_root.prc) OF
	MODE_ABSENT,
	MODE_INACTIVE:
		RETURN;
	MODE_TEST:
		RETURN;
END_CASE

ACTION _objects_manager:
IF	objects_initialization()
THEN
	axis_shadow_init(
		sim_mode:= SHADOW_SIMULATION_MODE_AUTOMATIC, 
		father:= csp_transfer_infeed_accu_waterfalladjust.axis, 
		process:= dbg_root.prc, 
		CONVERSION_this:= axis_shd);

	RETURN;
END_IF

IF	objects_running()
THEN
	axis_shadow_cycle(axis_shd);
END_IF
END_ACTION

END_PROGRAM

// ---- _Debug/dbg_csp_transfer_infeed_clamp.TcPOU

(********************* G.D S.p.A. - Technical Department ***********************************
This program has been generated automatically from Application Designer DE&F
********************************************************************************************)
PROGRAM dbg_csp_transfer_infeed_clamp
VAR
  extend_do_shd : digital_output_shadow;
  ls_retracted_di_shd : digital_input_shadow;
  ls_sact_shd : digital_actuator_shadow;
  os_retracted_di_shd : digital_input_shadow;
  os_sact_shd : digital_actuator_shadow;
END_VAR

_objects_manager();

IF	g_application_status <> APPLICATION_STATUS_RUNNING
THEN
	RETURN;
END_IF

CASE process_get_mode(CONVERSION_this := dbg_root.prc) OF
	MODE_ABSENT,
	MODE_INACTIVE:
		RETURN;
	MODE_TEST:
		RETURN;
END_CASE

ACTION _objects_manager:
IF	objects_initialization()
THEN
	digital_output_shadow_init(
		sim_mode:= SHADOW_SIMULATION_MODE_AUTOMATIC, 
		father:= csp_transfer_infeed_clamp.extend_do, 
		process:= dbg_root.prc, 
		CONVERSION_this:= extend_do_shd);

	digital_input_shadow_init(
		sim_mode:= SHADOW_SIMULATION_MODE_AUTOMATIC, 
		father:= csp_transfer_infeed_clamp.ls_retracted_di, 
		process:= dbg_root.prc, 
		CONVERSION_this:= ls_retracted_di_shd);

	digital_actuator_shadow_init(
		sim_mode:= SHADOW_SIMULATION_MODE_AUTOMATIC, 
		father:= csp_transfer_infeed_clamp.ls_sact, 
		process:= dbg_root.prc, 
		CONVERSION_this:= ls_sact_shd);

	digital_input_shadow_init(
		sim_mode:= SHADOW_SIMULATION_MODE_AUTOMATIC, 
		father:= csp_transfer_infeed_clamp.os_retracted_di, 
		process:= dbg_root.prc, 
		CONVERSION_this:= os_retracted_di_shd);

	digital_actuator_shadow_init(
		sim_mode:= SHADOW_SIMULATION_MODE_AUTOMATIC, 
		father:= csp_transfer_infeed_clamp.os_sact, 
		process:= dbg_root.prc, 
		CONVERSION_this:= os_sact_shd);

	RETURN;
END_IF

IF	objects_running()
THEN
	digital_output_shadow_cycle(extend_do_shd);
	digital_input_shadow_cycle(ls_retracted_di_shd);
	digital_actuator_shadow_cycle(ls_sact_shd);
	digital_input_shadow_cycle(os_retracted_di_shd);
	digital_actuator_shadow_cycle(os_sact_shd);
END_IF
END_ACTION

END_PROGRAM

// ---- _Debug/dbg_csp_transfer_infeed_metering_belt.TcPOU

(********************* G.D S.p.A. - Technical Department ***********************************
This program has been generated automatically from Application Designer DE&F
********************************************************************************************)
PROGRAM dbg_csp_transfer_infeed_metering_belt
VAR
  axis_shd : axis_shadow;
END_VAR

_objects_manager();

IF	g_application_status <> APPLICATION_STATUS_RUNNING
THEN
	RETURN;
END_IF

CASE process_get_mode(CONVERSION_this := dbg_root.prc) OF
	MODE_ABSENT,
	MODE_INACTIVE:
		RETURN;
	MODE_TEST:
		RETURN;
END_CASE

ACTION _objects_manager:
IF	objects_initialization()
THEN
	axis_shadow_init(
		sim_mode:= SHADOW_SIMULATION_MODE_AUTOMATIC, 
		father:= csp_transfer_infeed_metering_belt.axis, 
		process:= dbg_root.prc, 
		CONVERSION_this:= axis_shd);

	RETURN;
END_IF

IF	objects_running()
THEN
	axis_shadow_cycle(axis_shd);
END_IF
END_ACTION

END_PROGRAM

// ---- _Debug/dbg_csp_transfer_infeed_metering_jam.TcPOU

(********************* G.D S.p.A. - Technical Department ***********************************
This program has been generated automatically from Application Designer DE&F
********************************************************************************************)
PROGRAM dbg_csp_transfer_infeed_metering_jam
VAR
  jam_di_shd : digital_input_shadow;
  jam_sensor_on_dchk_shd : digital_check_shadow;
END_VAR

_objects_manager();

IF	g_application_status <> APPLICATION_STATUS_RUNNING
THEN
	RETURN;
END_IF

CASE process_get_mode(CONVERSION_this := dbg_root.prc) OF
	MODE_ABSENT,
	MODE_INACTIVE:
		RETURN;
	MODE_TEST:
		RETURN;
END_CASE

ACTION _objects_manager:
IF	objects_initialization()
THEN
	digital_input_shadow_init(
		sim_mode:= SHADOW_SIMULATION_MODE_AUTOMATIC, 
		father:= csp_transfer_infeed_metering_jam.jam_di, 
		process:= dbg_root.prc, 
		CONVERSION_this:= jam_di_shd);

	digital_check_shadow_init(
		sim_mode:= SHADOW_SIMULATION_MODE_AUTOMATIC, 
		father:= csp_transfer_infeed_metering_jam.jam_sensor_on_dchk, 
		process:= dbg_root.prc, 
		CONVERSION_this:= jam_sensor_on_dchk_shd);

	RETURN;
END_IF

IF	objects_running()
THEN
	digital_input_shadow_cycle(jam_di_shd);
	digital_check_shadow_cycle(jam_sensor_on_dchk_shd);
END_IF
END_ACTION

END_PROGRAM

// ---- _Debug/dbg_csp_transfer_infeed_reject_highload.TcPOU

(********************* G.D S.p.A. - Technical Department ***********************************
This program has been generated automatically from Application Designer DE&F
********************************************************************************************)
PROGRAM dbg_csp_transfer_infeed_reject_highload
VAR
  high_achk_shd : analog_check_shadow;
  high_ai_shd : analog_input_shadow;
END_VAR

_objects_manager();

IF	g_application_status <> APPLICATION_STATUS_RUNNING
THEN
	RETURN;
END_IF

CASE process_get_mode(CONVERSION_this := dbg_root.prc) OF
	MODE_ABSENT,
	MODE_INACTIVE:
		RETURN;
	MODE_TEST:
		RETURN;
END_CASE

ACTION _objects_manager:
IF	objects_initialization()
THEN
	analog_check_shadow_init(
		sim_mode:= SHADOW_SIMULATION_MODE_AUTOMATIC, 
		father:= csp_transfer_infeed_reject_highload.high_achk, 
		process:= dbg_root.prc, 
		CONVERSION_this:= high_achk_shd);

	analog_input_shadow_init(
		sim_mode:= SHADOW_SIMULATION_MODE_AUTOMATIC, 
		father:= csp_transfer_infeed_reject_highload.high_ai, 
		process:= dbg_root.prc, 
		CONVERSION_this:= high_ai_shd);

	RETURN;
END_IF

IF	objects_running()
THEN
	analog_check_shadow_cycle(high_achk_shd);
	analog_input_shadow_cycle(high_ai_shd);
END_IF
END_ACTION

END_PROGRAM

// ---- _Debug/dbg_csp_transfer_infeed_reject_pusher.TcPOU

(********************* G.D S.p.A. - Technical Department ***********************************
This program has been generated automatically from Application Designer DE&F
********************************************************************************************)
PROGRAM dbg_csp_transfer_infeed_reject_pusher
VAR
  axis_shd : axis_shadow;
END_VAR

_objects_manager();

IF	g_application_status <> APPLICATION_STATUS_RUNNING
THEN
	RETURN;
END_IF

CASE process_get_mode(CONVERSION_this := dbg_root.prc) OF
	MODE_ABSENT,
	MODE_INACTIVE:
		RETURN;
	MODE_TEST:
		RETURN;
END_CASE

ACTION _objects_manager:
IF	objects_initialization()
THEN
	axis_shadow_init(
		sim_mode:= SHADOW_SIMULATION_MODE_AUTOMATIC, 
		father:= csp_transfer_infeed_reject_pusher.axis, 
		process:= dbg_root.prc, 
		CONVERSION_this:= axis_shd);

	RETURN;
END_IF

IF	objects_running()
THEN
	axis_shadow_cycle(axis_shd);
END_IF
END_ACTION

END_PROGRAM

// ---- _Debug/dbg_csp_transfer_infeed_reject_virtualmaster.TcPOU

(********************* G.D S.p.A. - Technical Department ***********************************
This program has been generated automatically from Application Designer DE&F
********************************************************************************************)
PROGRAM dbg_csp_transfer_infeed_reject_virtualmaster
VAR
  axis_shd : axis_shadow;
END_VAR

_objects_manager();

IF	g_application_status <> APPLICATION_STATUS_RUNNING
THEN
	RETURN;
END_IF

CASE process_get_mode(CONVERSION_this := dbg_root.prc) OF
	MODE_ABSENT,
	MODE_INACTIVE:
		RETURN;
	MODE_TEST:
		RETURN;
END_CASE

ACTION _objects_manager:
IF	objects_initialization()
THEN
	axis_shadow_init(
		sim_mode:= SHADOW_SIMULATION_MODE_AUTOMATIC, 
		father:= csp_transfer_infeed_reject_virtualmaster.axis, 
		process:= dbg_root.prc, 
		CONVERSION_this:= axis_shd);

	RETURN;
END_IF

IF	objects_running()
THEN
	axis_shadow_cycle(axis_shd);
END_IF
END_ACTION

END_PROGRAM

// ---- _Debug/dbg_csp_transfer_infeed_waterfall_belt.TcPOU

(********************* G.D S.p.A. - Technical Department ***********************************
This program has been generated automatically from Application Designer DE&F
********************************************************************************************)
PROGRAM dbg_csp_transfer_infeed_waterfall_belt
VAR
  axis_shd : axis_shadow;
END_VAR

_objects_manager();

IF	g_application_status <> APPLICATION_STATUS_RUNNING
THEN
	RETURN;
END_IF

CASE process_get_mode(CONVERSION_this := dbg_root.prc) OF
	MODE_ABSENT,
	MODE_INACTIVE:
		RETURN;
	MODE_TEST:
		RETURN;
END_CASE

ACTION _objects_manager:
IF	objects_initialization()
THEN
	axis_shadow_init(
		sim_mode:= SHADOW_SIMULATION_MODE_AUTOMATIC, 
		father:= csp_transfer_infeed_waterfall_belt.axis, 
		process:= dbg_root.prc, 
		CONVERSION_this:= axis_shd);

	RETURN;
END_IF

IF	objects_running()
THEN
	axis_shadow_cycle(axis_shd);
END_IF
END_ACTION

END_PROGRAM

// ---- _Debug/dbg_csp_transfer_main_safety_accuchange.TcPOU

(********************* G.D S.p.A. - Technical Department ***********************************
This program has been generated automatically from Application Designer DE&F
********************************************************************************************)
PROGRAM dbg_csp_transfer_main_safety_accuchange
VAR
  sis_shd : safety_integrated_series_shadow;
END_VAR

_objects_manager();

IF	g_application_status <> APPLICATION_STATUS_RUNNING
THEN
	RETURN;
END_IF

CASE process_get_mode(CONVERSION_this := dbg_root.prc) OF
	MODE_ABSENT,
	MODE_INACTIVE:
		RETURN;
	MODE_TEST:
		RETURN;
END_CASE

ACTION _objects_manager:
IF	objects_initialization()
THEN
	safety_integrated_series_shadow_init(
		sim_mode:= SHADOW_SIMULATION_MODE_AUTOMATIC, 
		father:= csp_transfer_main_safety_accuchange.sis, 
		process:= dbg_root.prc, 
		CONVERSION_this:= sis_shd);

	RETURN;
END_IF

IF	objects_running()
THEN
	safety_integrated_series_shadow_cycle(sis_shd);
END_IF
END_ACTION

END_PROGRAM

// ---- _Debug/dbg_csp_transfer_main_safety_drives_commonconfiguration.TcPOU

(********************* G.D S.p.A. - Technical Department ***********************************
This program has been generated automatically from Application Designer DE&F
********************************************************************************************)
PROGRAM dbg_csp_transfer_main_safety_drives_commonconfiguration
VAR
  rack_smes_sis_shd : safety_integrated_series_shadow;
  standalone_smes_sis_shd : safety_integrated_series_shadow;
END_VAR

_objects_manager();

IF	g_application_status <> APPLICATION_STATUS_RUNNING
THEN
	RETURN;
END_IF

CASE process_get_mode(CONVERSION_this := dbg_root.prc) OF
	MODE_ABSENT,
	MODE_INACTIVE:
		RETURN;
	MODE_TEST:
		RETURN;
END_CASE

ACTION _objects_manager:
IF	objects_initialization()
THEN
	safety_integrated_series_shadow_init(
		sim_mode:= SHADOW_SIMULATION_MODE_AUTOMATIC, 
		father:= csp_transfer_main_safety_drives_commonconfiguration.rack_smes_sis, 
		process:= dbg_root.prc, 
		CONVERSION_this:= rack_smes_sis_shd);

	safety_integrated_series_shadow_init(
		sim_mode:= SHADOW_SIMULATION_MODE_AUTOMATIC, 
		father:= csp_transfer_main_safety_drives_commonconfiguration.standalone_smes_sis, 
		process:= dbg_root.prc, 
		CONVERSION_this:= standalone_smes_sis_shd);

	RETURN;
END_IF

IF	objects_running()
THEN
	safety_integrated_series_shadow_cycle(rack_smes_sis_shd);
	safety_integrated_series_shadow_cycle(standalone_smes_sis_shd);
END_IF
END_ACTION

END_PROGRAM

// ---- _Debug/dbg_csp_transfer_main_safety_drives_ps41020.TcPOU

(********************* G.D S.p.A. - Technical Department ***********************************
This program has been generated automatically from Application Designer DE&F
********************************************************************************************)
PROGRAM dbg_csp_transfer_main_safety_drives_ps41020
VAR
  sis_shd : safety_integrated_series_shadow;
END_VAR

_objects_manager();

IF	g_application_status <> APPLICATION_STATUS_RUNNING
THEN
	RETURN;
END_IF

CASE process_get_mode(CONVERSION_this := dbg_root.prc) OF
	MODE_ABSENT,
	MODE_INACTIVE:
		RETURN;
	MODE_TEST:
		RETURN;
END_CASE

ACTION _objects_manager:
IF	objects_initialization()
THEN
	safety_integrated_series_shadow_init(
		sim_mode:= SHADOW_SIMULATION_MODE_AUTOMATIC, 
		father:= csp_transfer_main_safety_drives_ps41020.sis, 
		process:= dbg_root.prc, 
		CONVERSION_this:= sis_shd);

	RETURN;
END_IF

IF	objects_running()
THEN
	safety_integrated_series_shadow_cycle(sis_shd);
END_IF
END_ACTION

END_PROGRAM

// ---- _Debug/dbg_csp_transfer_main_safety_drives_sd41100.TcPOU

(********************* G.D S.p.A. - Technical Department ***********************************
This program has been generated automatically from Application Designer DE&F
********************************************************************************************)
PROGRAM dbg_csp_transfer_main_safety_drives_sd41100
VAR
  cha_smes_sis_shd : safety_integrated_series_shadow;
  chb_smes_sis_shd : safety_integrated_series_shadow;
END_VAR

_objects_manager();

IF	g_application_status <> APPLICATION_STATUS_RUNNING
THEN
	RETURN;
END_IF

CASE process_get_mode(CONVERSION_this := dbg_root.prc) OF
	MODE_ABSENT,
	MODE_INACTIVE:
		RETURN;
	MODE_TEST:
		RETURN;
END_CASE

ACTION _objects_manager:
IF	objects_initialization()
THEN
	safety_integrated_series_shadow_init(
		sim_mode:= SHADOW_SIMULATION_MODE_AUTOMATIC, 
		father:= csp_transfer_main_safety_drives_sd41100.cha_smes_sis, 
		process:= dbg_root.prc, 
		CONVERSION_this:= cha_smes_sis_shd);

	safety_integrated_series_shadow_init(
		sim_mode:= SHADOW_SIMULATION_MODE_AUTOMATIC, 
		father:= csp_transfer_main_safety_drives_sd41100.chb_smes_sis, 
		process:= dbg_root.prc, 
		CONVERSION_this:= chb_smes_sis_shd);

	RETURN;
END_IF

IF	objects_running()
THEN
	safety_integrated_series_shadow_cycle(cha_smes_sis_shd);
	safety_integrated_series_shadow_cycle(chb_smes_sis_shd);
END_IF
END_ACTION

END_PROGRAM

// ---- _Debug/dbg_csp_transfer_main_safety_drives_sd41200.TcPOU

(********************* G.D S.p.A. - Technical Department ***********************************
This program has been generated automatically from Application Designer DE&F
********************************************************************************************)
PROGRAM dbg_csp_transfer_main_safety_drives_sd41200
VAR
  cha_smes_sis_shd : safety_integrated_series_shadow;
  chb_smes_sis_shd : safety_integrated_series_shadow;
END_VAR

_objects_manager();

IF	g_application_status <> APPLICATION_STATUS_RUNNING
THEN
	RETURN;
END_IF

CASE process_get_mode(CONVERSION_this := dbg_root.prc) OF
	MODE_ABSENT,
	MODE_INACTIVE:
		RETURN;
	MODE_TEST:
		RETURN;
END_CASE

ACTION _objects_manager:
IF	objects_initialization()
THEN
	safety_integrated_series_shadow_init(
		sim_mode:= SHADOW_SIMULATION_MODE_AUTOMATIC, 
		father:= csp_transfer_main_safety_drives_sd41200.cha_smes_sis, 
		process:= dbg_root.prc, 
		CONVERSION_this:= cha_smes_sis_shd);

	safety_integrated_series_shadow_init(
		sim_mode:= SHADOW_SIMULATION_MODE_AUTOMATIC, 
		father:= csp_transfer_main_safety_drives_sd41200.chb_smes_sis, 
		process:= dbg_root.prc, 
		CONVERSION_this:= chb_smes_sis_shd);

	RETURN;
END_IF

IF	objects_running()
THEN
	safety_integrated_series_shadow_cycle(cha_smes_sis_shd);
	safety_integrated_series_shadow_cycle(chb_smes_sis_shd);
END_IF
END_ACTION

END_PROGRAM

// ---- _Debug/dbg_csp_transfer_main_safety_drives_sd41300.TcPOU

(********************* G.D S.p.A. - Technical Department ***********************************
This program has been generated automatically from Application Designer DE&F
********************************************************************************************)
PROGRAM dbg_csp_transfer_main_safety_drives_sd41300
VAR
  cha_smes_sis_shd : safety_integrated_series_shadow;
  chb_smes_sis_shd : safety_integrated_series_shadow;
END_VAR

_objects_manager();

IF	g_application_status <> APPLICATION_STATUS_RUNNING
THEN
	RETURN;
END_IF

CASE process_get_mode(CONVERSION_this := dbg_root.prc) OF
	MODE_ABSENT,
	MODE_INACTIVE:
		RETURN;
	MODE_TEST:
		RETURN;
END_CASE

ACTION _objects_manager:
IF	objects_initialization()
THEN
	safety_integrated_series_shadow_init(
		sim_mode:= SHADOW_SIMULATION_MODE_AUTOMATIC, 
		father:= csp_transfer_main_safety_drives_sd41300.cha_smes_sis, 
		process:= dbg_root.prc, 
		CONVERSION_this:= cha_smes_sis_shd);

	safety_integrated_series_shadow_init(
		sim_mode:= SHADOW_SIMULATION_MODE_AUTOMATIC, 
		father:= csp_transfer_main_safety_drives_sd41300.chb_smes_sis, 
		process:= dbg_root.prc, 
		CONVERSION_this:= chb_smes_sis_shd);

	RETURN;
END_IF

IF	objects_running()
THEN
	safety_integrated_series_shadow_cycle(cha_smes_sis_shd);
	safety_integrated_series_shadow_cycle(chb_smes_sis_shd);
END_IF
END_ACTION

END_PROGRAM

// ---- _Debug/dbg_csp_transfer_main_safety_drives_sd41400.TcPOU

(********************* G.D S.p.A. - Technical Department ***********************************
This program has been generated automatically from Application Designer DE&F
********************************************************************************************)
PROGRAM dbg_csp_transfer_main_safety_drives_sd41400
VAR
  cha_smes_sis_shd : safety_integrated_series_shadow;
  chb_smes_sis_shd : safety_integrated_series_shadow;
END_VAR

_objects_manager();

IF	g_application_status <> APPLICATION_STATUS_RUNNING
THEN
	RETURN;
END_IF

CASE process_get_mode(CONVERSION_this := dbg_root.prc) OF
	MODE_ABSENT,
	MODE_INACTIVE:
		RETURN;
	MODE_TEST:
		RETURN;
END_CASE

ACTION _objects_manager:
IF	objects_initialization()
THEN
	safety_integrated_series_shadow_init(
		sim_mode:= SHADOW_SIMULATION_MODE_AUTOMATIC, 
		father:= csp_transfer_main_safety_drives_sd41400.cha_smes_sis, 
		process:= dbg_root.prc, 
		CONVERSION_this:= cha_smes_sis_shd);

	safety_integrated_series_shadow_init(
		sim_mode:= SHADOW_SIMULATION_MODE_AUTOMATIC, 
		father:= csp_transfer_main_safety_drives_sd41400.chb_smes_sis, 
		process:= dbg_root.prc, 
		CONVERSION_this:= chb_smes_sis_shd);

	RETURN;
END_IF

IF	objects_running()
THEN
	safety_integrated_series_shadow_cycle(cha_smes_sis_shd);
	safety_integrated_series_shadow_cycle(chb_smes_sis_shd);
END_IF
END_ACTION

END_PROGRAM

// ---- _Debug/dbg_csp_transfer_main_safety_drives_sd41500.TcPOU

(********************* G.D S.p.A. - Technical Department ***********************************
This program has been generated automatically from Application Designer DE&F
********************************************************************************************)
PROGRAM dbg_csp_transfer_main_safety_drives_sd41500
VAR
  cha_smes_sis_shd : safety_integrated_series_shadow;
  chb_smes_sis_shd : safety_integrated_series_shadow;
END_VAR

_objects_manager();

IF	g_application_status <> APPLICATION_STATUS_RUNNING
THEN
	RETURN;
END_IF

CASE process_get_mode(CONVERSION_this := dbg_root.prc) OF
	MODE_ABSENT,
	MODE_INACTIVE:
		RETURN;
	MODE_TEST:
		RETURN;
END_CASE

ACTION _objects_manager:
IF	objects_initialization()
THEN
	safety_integrated_series_shadow_init(
		sim_mode:= SHADOW_SIMULATION_MODE_AUTOMATIC, 
		father:= csp_transfer_main_safety_drives_sd41500.cha_smes_sis, 
		process:= dbg_root.prc, 
		CONVERSION_this:= cha_smes_sis_shd);

	safety_integrated_series_shadow_init(
		sim_mode:= SHADOW_SIMULATION_MODE_AUTOMATIC, 
		father:= csp_transfer_main_safety_drives_sd41500.chb_smes_sis, 
		process:= dbg_root.prc, 
		CONVERSION_this:= chb_smes_sis_shd);

	RETURN;
END_IF

IF	objects_running()
THEN
	safety_integrated_series_shadow_cycle(cha_smes_sis_shd);
	safety_integrated_series_shadow_cycle(chb_smes_sis_shd);
END_IF
END_ACTION

END_PROGRAM

// ---- _Debug/dbg_csp_transfer_main_safety_drives_sd41600.TcPOU

(********************* G.D S.p.A. - Technical Department ***********************************
This program has been generated automatically from Application Designer DE&F
********************************************************************************************)
PROGRAM dbg_csp_transfer_main_safety_drives_sd41600
VAR
  cha_smes_sis_shd : safety_integrated_series_shadow;
  chb_smes_sis_shd : safety_integrated_series_shadow;
END_VAR

_objects_manager();

IF	g_application_status <> APPLICATION_STATUS_RUNNING
THEN
	RETURN;
END_IF

CASE process_get_mode(CONVERSION_this := dbg_root.prc) OF
	MODE_ABSENT,
	MODE_INACTIVE:
		RETURN;
	MODE_TEST:
		RETURN;
END_CASE

ACTION _objects_manager:
IF	objects_initialization()
THEN
	safety_integrated_series_shadow_init(
		sim_mode:= SHADOW_SIMULATION_MODE_AUTOMATIC, 
		father:= csp_transfer_main_safety_drives_sd41600.cha_smes_sis, 
		process:= dbg_root.prc, 
		CONVERSION_this:= cha_smes_sis_shd);

	safety_integrated_series_shadow_init(
		sim_mode:= SHADOW_SIMULATION_MODE_AUTOMATIC, 
		father:= csp_transfer_main_safety_drives_sd41600.chb_smes_sis, 
		process:= dbg_root.prc, 
		CONVERSION_this:= chb_smes_sis_shd);

	RETURN;
END_IF

IF	objects_running()
THEN
	safety_integrated_series_shadow_cycle(cha_smes_sis_shd);
	safety_integrated_series_shadow_cycle(chb_smes_sis_shd);
END_IF
END_ACTION

END_PROGRAM

// ---- _Debug/dbg_csp_transfer_main_safety_drives_sd41700.TcPOU

(********************* G.D S.p.A. - Technical Department ***********************************
This program has been generated automatically from Application Designer DE&F
********************************************************************************************)
PROGRAM dbg_csp_transfer_main_safety_drives_sd41700
VAR
  cha_smes_sis_shd : safety_integrated_series_shadow;
  chb_smes_sis_shd : safety_integrated_series_shadow;
END_VAR

_objects_manager();

IF	g_application_status <> APPLICATION_STATUS_RUNNING
THEN
	RETURN;
END_IF

CASE process_get_mode(CONVERSION_this := dbg_root.prc) OF
	MODE_ABSENT,
	MODE_INACTIVE:
		RETURN;
	MODE_TEST:
		RETURN;
END_CASE

ACTION _objects_manager:
IF	objects_initialization()
THEN
	safety_integrated_series_shadow_init(
		sim_mode:= SHADOW_SIMULATION_MODE_AUTOMATIC, 
		father:= csp_transfer_main_safety_drives_sd41700.cha_smes_sis, 
		process:= dbg_root.prc, 
		CONVERSION_this:= cha_smes_sis_shd);

	safety_integrated_series_shadow_init(
		sim_mode:= SHADOW_SIMULATION_MODE_AUTOMATIC, 
		father:= csp_transfer_main_safety_drives_sd41700.chb_smes_sis, 
		process:= dbg_root.prc, 
		CONVERSION_this:= chb_smes_sis_shd);

	RETURN;
END_IF

IF	objects_running()
THEN
	safety_integrated_series_shadow_cycle(cha_smes_sis_shd);
	safety_integrated_series_shadow_cycle(chb_smes_sis_shd);
END_IF
END_ACTION

END_PROGRAM

// ---- _Debug/dbg_csp_transfer_main_safety_emergency.TcPOU

(********************* G.D S.p.A. - Technical Department ***********************************
This program has been generated automatically from Application Designer DE&F
********************************************************************************************)
PROGRAM dbg_csp_transfer_main_safety_emergency
VAR
  delayed_sis_shd : safety_integrated_series_shadow;
  hmi_button_lamp_do_shd : digital_output_shadow;
  hmi_button_sio_shd : safety_integrated_object_shadow;
  sis_shd : safety_integrated_series_shadow;
END_VAR

_objects_manager();

IF	g_application_status <> APPLICATION_STATUS_RUNNING
THEN
	RETURN;
END_IF

CASE process_get_mode(CONVERSION_this := dbg_root.prc) OF
	MODE_ABSENT,
	MODE_INACTIVE:
		RETURN;
	MODE_TEST:
		RETURN;
END_CASE

IF csp_transfer_main_services_pushbuttons.emergency_open_pressed
    THEN
        siss_open_series(sis_shd);
    ELSIF csp_transfer_main_services_pushbuttons.emergency_close_pressed
        THEN
        siss_close_series(sis_shd);
END_IF

ACTION _objects_manager:
IF	objects_initialization()
THEN
	safety_integrated_series_shadow_init(
		sim_mode:= SHADOW_SIMULATION_MODE_AUTOMATIC, 
		father:= csp_transfer_main_safety_emergency.delayed_sis, 
		process:= dbg_root.prc, 
		CONVERSION_this:= delayed_sis_shd);

	digital_output_shadow_init(
		sim_mode:= SHADOW_SIMULATION_MODE_AUTOMATIC, 
		father:= csp_transfer_main_safety_emergency.hmi_button_lamp_do, 
		process:= dbg_root.prc, 
		CONVERSION_this:= hmi_button_lamp_do_shd);

	safety_integrated_object_shadow_init(
		sim_mode:= SHADOW_SIMULATION_MODE_AUTOMATIC, 
		father:= csp_transfer_main_safety_emergency.hmi_button_sio, 
		process:= dbg_root.prc, 
		CONVERSION_this:= hmi_button_sio_shd);

	safety_integrated_series_shadow_init(
		sim_mode:= SHADOW_SIMULATION_MODE_AUTOMATIC, 
		father:= csp_transfer_main_safety_emergency.sis, 
		process:= dbg_root.prc, 
		CONVERSION_this:= sis_shd);

	RETURN;
END_IF

IF	objects_running()
THEN
	safety_integrated_series_shadow_cycle(delayed_sis_shd);
	digital_output_shadow_cycle(hmi_button_lamp_do_shd);
	safety_integrated_object_shadow_cycle(hmi_button_sio_shd);
	safety_integrated_series_shadow_cycle(sis_shd);
END_IF
END_ACTION

END_PROGRAM

// ---- _Debug/dbg_csp_transfer_main_safety_guards.TcPOU

(********************* G.D S.p.A. - Technical Department ***********************************
This program has been generated automatically from Application Designer DE&F
********************************************************************************************)
PROGRAM dbg_csp_transfer_main_safety_guards
VAR
  delayed_sis_shd : safety_integrated_series_shadow;
  sio_door_3_shd : safety_integrated_object_shadow;
  sio_door_4_shd : safety_integrated_object_shadow;
  sio_door_5_shd : safety_integrated_object_shadow;
  sio_door_6_shd : safety_integrated_object_shadow;
  sio_door_7_shd : safety_integrated_object_shadow;
  sio_door_8_shd : safety_integrated_object_shadow;
  sis_shd : safety_integrated_series_shadow;
END_VAR

_objects_manager();

IF	g_application_status <> APPLICATION_STATUS_RUNNING
THEN
	RETURN;
END_IF

CASE process_get_mode(CONVERSION_this := dbg_root.prc) OF
	MODE_ABSENT,
	MODE_INACTIVE:
		RETURN;
	MODE_TEST:
		RETURN;
END_CASE

ACTION _objects_manager:
IF	objects_initialization()
THEN
	safety_integrated_series_shadow_init(
		sim_mode:= SHADOW_SIMULATION_MODE_AUTOMATIC, 
		father:= csp_transfer_main_safety_guards.delayed_sis, 
		process:= dbg_root.prc, 
		CONVERSION_this:= delayed_sis_shd);

	safety_integrated_object_shadow_init(
		sim_mode:= SHADOW_SIMULATION_MODE_AUTOMATIC, 
		father:= csp_transfer_main_safety_guards.sio_door_3, 
		process:= dbg_root.prc, 
		CONVERSION_this:= sio_door_3_shd);

	safety_integrated_object_shadow_init(
		sim_mode:= SHADOW_SIMULATION_MODE_AUTOMATIC, 
		father:= csp_transfer_main_safety_guards.sio_door_4, 
		process:= dbg_root.prc, 
		CONVERSION_this:= sio_door_4_shd);

	safety_integrated_object_shadow_init(
		sim_mode:= SHADOW_SIMULATION_MODE_AUTOMATIC, 
		father:= csp_transfer_main_safety_guards.sio_door_5, 
		process:= dbg_root.prc, 
		CONVERSION_this:= sio_door_5_shd);

	safety_integrated_object_shadow_init(
		sim_mode:= SHADOW_SIMULATION_MODE_AUTOMATIC, 
		father:= csp_transfer_main_safety_guards.sio_door_6, 
		process:= dbg_root.prc, 
		CONVERSION_this:= sio_door_6_shd);

	safety_integrated_object_shadow_init(
		sim_mode:= SHADOW_SIMULATION_MODE_AUTOMATIC, 
		father:= csp_transfer_main_safety_guards.sio_door_7, 
		process:= dbg_root.prc, 
		CONVERSION_this:= sio_door_7_shd);

	safety_integrated_object_shadow_init(
		sim_mode:= SHADOW_SIMULATION_MODE_AUTOMATIC, 
		father:= csp_transfer_main_safety_guards.sio_door_8, 
		process:= dbg_root.prc, 
		CONVERSION_this:= sio_door_8_shd);

	safety_integrated_series_shadow_init(
		sim_mode:= SHADOW_SIMULATION_MODE_AUTOMATIC, 
		father:= csp_transfer_main_safety_guards.sis, 
		process:= dbg_root.prc, 
		CONVERSION_this:= sis_shd);

	RETURN;
END_IF

IF	objects_running()
THEN
	safety_integrated_series_shadow_cycle(delayed_sis_shd);
	safety_integrated_object_shadow_cycle(sio_door_3_shd);
	safety_integrated_object_shadow_cycle(sio_door_4_shd);
	safety_integrated_object_shadow_cycle(sio_door_5_shd);
	safety_integrated_object_shadow_cycle(sio_door_6_shd);
	safety_integrated_object_shadow_cycle(sio_door_7_shd);
	safety_integrated_object_shadow_cycle(sio_door_8_shd);
	safety_integrated_series_shadow_cycle(sis_shd);
END_IF
END_ACTION

END_PROGRAM

// ---- _Debug/dbg_csp_transfer_main_safety_token.TcPOU

(********************* G.D S.p.A. - Technical Department ***********************************
This program has been generated automatically from Application Designer DE&F
********************************************************************************************)
PROGRAM dbg_csp_transfer_main_safety_token
VAR
  sio_shd : safety_integrated_object_shadow;
  sis_shd : safety_integrated_series_shadow;
END_VAR

_objects_manager();

IF	g_application_status <> APPLICATION_STATUS_RUNNING
THEN
	RETURN;
END_IF

CASE process_get_mode(CONVERSION_this := dbg_root.prc) OF
	MODE_ABSENT,
	MODE_INACTIVE:
		RETURN;
	MODE_TEST:
		RETURN;
END_CASE

ACTION _objects_manager:
IF	objects_initialization()
THEN
	safety_integrated_object_shadow_init(
		sim_mode:= SHADOW_SIMULATION_MODE_AUTOMATIC, 
		father:= csp_transfer_main_safety_token.sio, 
		process:= dbg_root.prc, 
		CONVERSION_this:= sio_shd);

	safety_integrated_series_shadow_init(
		sim_mode:= SHADOW_SIMULATION_MODE_AUTOMATIC, 
		father:= csp_transfer_main_safety_token.sis, 
		process:= dbg_root.prc, 
		CONVERSION_this:= sis_shd);

	RETURN;
END_IF

IF	objects_running()
THEN
	safety_integrated_object_shadow_cycle(sio_shd);
	safety_integrated_series_shadow_cycle(sis_shd);
END_IF
END_ACTION

END_PROGRAM

// ---- _Debug/dbg_csp_transfer_main_services.TcPOU

(********************* G.D S.p.A. - Technical Department ***********************************
This program has been generated automatically from Application Designer DE&F
********************************************************************************************)
PROGRAM dbg_csp_transfer_main_services
VAR
  reset_output_test_shd : digital_output_shadow;
END_VAR

_objects_manager();

IF	g_application_status <> APPLICATION_STATUS_RUNNING
THEN
	RETURN;
END_IF

CASE process_get_mode(CONVERSION_this := dbg_root.prc) OF
	MODE_ABSENT,
	MODE_INACTIVE:
		RETURN;
	MODE_TEST:
		RETURN;
END_CASE

ACTION _objects_manager:
IF	objects_initialization()
THEN
	digital_output_shadow_init(
		sim_mode:= SHADOW_SIMULATION_MODE_AUTOMATIC, 
		father:= csp_transfer_main_services.reset_output_test, 
		process:= dbg_root.prc, 
		CONVERSION_this:= reset_output_test_shd);

	RETURN;
END_IF

IF	objects_running()
THEN
	digital_output_shadow_cycle(reset_output_test_shd);
END_IF
END_ACTION

END_PROGRAM

// ---- _Debug/dbg_csp_transfer_main_services_breakers.TcPOU

(********************* G.D S.p.A. - Technical Department ***********************************
This program has been generated automatically from Application Designer DE&F
********************************************************************************************)
PROGRAM dbg_csp_transfer_main_services_breakers
VAR
  psw1_monitor_dchk_shd : digital_check_shadow;
  psw1_monitor_di_shd : digital_input_shadow;
  psw2_monitor_dchk_shd : digital_check_shadow;
  psw2_monitor_di_shd : digital_input_shadow;
  psw3_monitor_dchk_shd : digital_check_shadow;
  psw3_monitor_di_shd : digital_input_shadow;
  psw4_monitor_dchk_shd : digital_check_shadow;
  psw4_monitor_di_shd : digital_input_shadow;
  psw5_monitor_dchk_shd : digital_check_shadow;
  psw5_monitor_di_shd : digital_input_shadow;
  psw6_monitor_dchk_shd : digital_check_shadow;
  psw6_monitor_di_shd : digital_input_shadow;
END_VAR

_objects_manager();

IF	g_application_status <> APPLICATION_STATUS_RUNNING
THEN
	RETURN;
END_IF

CASE process_get_mode(CONVERSION_this := dbg_root.prc) OF
	MODE_ABSENT,
	MODE_INACTIVE:
		RETURN;
	MODE_TEST:
		RETURN;
END_CASE

ACTION _objects_manager:
IF	objects_initialization()
THEN
	digital_check_shadow_init(
		sim_mode:= SHADOW_SIMULATION_MODE_AUTOMATIC, 
		father:= csp_transfer_main_services_breakers.psw1_monitor_dchk, 
		process:= dbg_root.prc, 
		CONVERSION_this:= psw1_monitor_dchk_shd);

	digital_input_shadow_init(
		sim_mode:= SHADOW_SIMULATION_MODE_AUTOMATIC, 
		father:= csp_transfer_main_services_breakers.psw1_monitor_di, 
		process:= dbg_root.prc, 
		CONVERSION_this:= psw1_monitor_di_shd);

	digital_check_shadow_init(
		sim_mode:= SHADOW_SIMULATION_MODE_AUTOMATIC, 
		father:= csp_transfer_main_services_breakers.psw2_monitor_dchk, 
		process:= dbg_root.prc, 
		CONVERSION_this:= psw2_monitor_dchk_shd);

	digital_input_shadow_init(
		sim_mode:= SHADOW_SIMULATION_MODE_AUTOMATIC, 
		father:= csp_transfer_main_services_breakers.psw2_monitor_di, 
		process:= dbg_root.prc, 
		CONVERSION_this:= psw2_monitor_di_shd);

	digital_check_shadow_init(
		sim_mode:= SHADOW_SIMULATION_MODE_AUTOMATIC, 
		father:= csp_transfer_main_services_breakers.psw3_monitor_dchk, 
		process:= dbg_root.prc, 
		CONVERSION_this:= psw3_monitor_dchk_shd);

	digital_input_shadow_init(
		sim_mode:= SHADOW_SIMULATION_MODE_AUTOMATIC, 
		father:= csp_transfer_main_services_breakers.psw3_monitor_di, 
		process:= dbg_root.prc, 
		CONVERSION_this:= psw3_monitor_di_shd);

	digital_check_shadow_init(
		sim_mode:= SHADOW_SIMULATION_MODE_AUTOMATIC, 
		father:= csp_transfer_main_services_breakers.psw4_monitor_dchk, 
		process:= dbg_root.prc, 
		CONVERSION_this:= psw4_monitor_dchk_shd);

	digital_input_shadow_init(
		sim_mode:= SHADOW_SIMULATION_MODE_AUTOMATIC, 
		father:= csp_transfer_main_services_breakers.psw4_monitor_di, 
		process:= dbg_root.prc, 
		CONVERSION_this:= psw4_monitor_di_shd);

	digital_check_shadow_init(
		sim_mode:= SHADOW_SIMULATION_MODE_AUTOMATIC, 
		father:= csp_transfer_main_services_breakers.psw5_monitor_dchk, 
		process:= dbg_root.prc, 
		CONVERSION_this:= psw5_monitor_dchk_shd);

	digital_input_shadow_init(
		sim_mode:= SHADOW_SIMULATION_MODE_AUTOMATIC, 
		father:= csp_transfer_main_services_breakers.psw5_monitor_di, 
		process:= dbg_root.prc, 
		CONVERSION_this:= psw5_monitor_di_shd);

	digital_check_shadow_init(
		sim_mode:= SHADOW_SIMULATION_MODE_AUTOMATIC, 
		father:= csp_transfer_main_services_breakers.psw6_monitor_dchk, 
		process:= dbg_root.prc, 
		CONVERSION_this:= psw6_monitor_dchk_shd);

	digital_input_shadow_init(
		sim_mode:= SHADOW_SIMULATION_MODE_AUTOMATIC, 
		father:= csp_transfer_main_services_breakers.psw6_monitor_di, 
		process:= dbg_root.prc, 
		CONVERSION_this:= psw6_monitor_di_shd);

	RETURN;
END_IF

IF	objects_running()
THEN
	digital_check_shadow_cycle(psw1_monitor_dchk_shd);
	digital_input_shadow_cycle(psw1_monitor_di_shd);
	digital_check_shadow_cycle(psw2_monitor_dchk_shd);
	digital_input_shadow_cycle(psw2_monitor_di_shd);
	digital_check_shadow_cycle(psw3_monitor_dchk_shd);
	digital_input_shadow_cycle(psw3_monitor_di_shd);
	digital_check_shadow_cycle(psw4_monitor_dchk_shd);
	digital_input_shadow_cycle(psw4_monitor_di_shd);
	digital_check_shadow_cycle(psw5_monitor_dchk_shd);
	digital_input_shadow_cycle(psw5_monitor_di_shd);
	digital_check_shadow_cycle(psw6_monitor_dchk_shd);
	digital_input_shadow_cycle(psw6_monitor_di_shd);
END_IF
END_ACTION

END_PROGRAM

// ---- _Debug/dbg_csp_transfer_main_services_pushbuttons.TcPOU

(********************* G.D S.p.A. - Technical Department ***********************************
This program has been generated automatically from Application Designer DE&F
********************************************************************************************)
PROGRAM dbg_csp_transfer_main_services_pushbuttons
VAR
  emergency_close_di_shd : digital_input_shadow;
  emergency_close_lamp_do_shd : digital_output_shadow;
  emergency_open_di_shd : digital_input_shadow;
  emergency_open_lamp_do_shd : digital_output_shadow;
  reset_di_shd : digital_input_shadow;
  reset_lamp_do_shd : digital_output_shadow;
  start_di_shd : digital_input_shadow;
  start_lamp_do_shd : digital_output_shadow;
  stop_dchk_shd : digital_check_shadow;
  stop_di_shd : digital_input_shadow;
  stop_lamp_do_shd : digital_output_shadow;
END_VAR

_objects_manager();

IF	g_application_status <> APPLICATION_STATUS_RUNNING
THEN
	RETURN;
END_IF

CASE process_get_mode(CONVERSION_this := dbg_root.prc) OF
	MODE_ABSENT,
	MODE_INACTIVE:
		RETURN;
	MODE_TEST:
		RETURN;
END_CASE

ACTION _objects_manager:
IF	objects_initialization()
THEN
	digital_input_shadow_init(
		sim_mode:= SHADOW_SIMULATION_MODE_AUTOMATIC, 
		father:= csp_transfer_main_services_pushbuttons.emergency_close_di, 
		process:= dbg_root.prc, 
		CONVERSION_this:= emergency_close_di_shd);

	digital_output_shadow_init(
		sim_mode:= SHADOW_SIMULATION_MODE_AUTOMATIC, 
		father:= csp_transfer_main_services_pushbuttons.emergency_close_lamp_do, 
		process:= dbg_root.prc, 
		CONVERSION_this:= emergency_close_lamp_do_shd);

	digital_input_shadow_init(
		sim_mode:= SHADOW_SIMULATION_MODE_AUTOMATIC, 
		father:= csp_transfer_main_services_pushbuttons.emergency_open_di, 
		process:= dbg_root.prc, 
		CONVERSION_this:= emergency_open_di_shd);

	digital_output_shadow_init(
		sim_mode:= SHADOW_SIMULATION_MODE_AUTOMATIC, 
		father:= csp_transfer_main_services_pushbuttons.emergency_open_lamp_do, 
		process:= dbg_root.prc, 
		CONVERSION_this:= emergency_open_lamp_do_shd);

	digital_input_shadow_init(
		sim_mode:= SHADOW_SIMULATION_MODE_AUTOMATIC, 
		father:= csp_transfer_main_services_pushbuttons.reset_di, 
		process:= dbg_root.prc, 
		CONVERSION_this:= reset_di_shd);

	digital_output_shadow_init(
		sim_mode:= SHADOW_SIMULATION_MODE_AUTOMATIC, 
		father:= csp_transfer_main_services_pushbuttons.reset_lamp_do, 
		process:= dbg_root.prc, 
		CONVERSION_this:= reset_lamp_do_shd);

	digital_input_shadow_init(
		sim_mode:= SHADOW_SIMULATION_MODE_AUTOMATIC, 
		father:= csp_transfer_main_services_pushbuttons.start_di, 
		process:= dbg_root.prc, 
		CONVERSION_this:= start_di_shd);

	digital_output_shadow_init(
		sim_mode:= SHADOW_SIMULATION_MODE_AUTOMATIC, 
		father:= csp_transfer_main_services_pushbuttons.start_lamp_do, 
		process:= dbg_root.prc, 
		CONVERSION_this:= start_lamp_do_shd);

	digital_check_shadow_init(
		sim_mode:= SHADOW_SIMULATION_MODE_AUTOMATIC, 
		father:= csp_transfer_main_services_pushbuttons.stop_dchk, 
		process:= dbg_root.prc, 
		CONVERSION_this:= stop_dchk_shd);

	digital_input_shadow_init(
		sim_mode:= SHADOW_SIMULATION_MODE_AUTOMATIC, 
		father:= csp_transfer_main_services_pushbuttons.stop_di, 
		process:= dbg_root.prc, 
		CONVERSION_this:= stop_di_shd);

	digital_output_shadow_init(
		sim_mode:= SHADOW_SIMULATION_MODE_AUTOMATIC, 
		father:= csp_transfer_main_services_pushbuttons.stop_lamp_do, 
		process:= dbg_root.prc, 
		CONVERSION_this:= stop_lamp_do_shd);

	RETURN;
END_IF

IF	objects_running()
THEN
	digital_input_shadow_cycle(emergency_close_di_shd);
	digital_output_shadow_cycle(emergency_close_lamp_do_shd);
	digital_input_shadow_cycle(emergency_open_di_shd);
	digital_output_shadow_cycle(emergency_open_lamp_do_shd);
	digital_input_shadow_cycle(reset_di_shd);
	digital_output_shadow_cycle(reset_lamp_do_shd);
	digital_input_shadow_cycle(start_di_shd);
	digital_output_shadow_cycle(start_lamp_do_shd);
	digital_check_shadow_cycle(stop_dchk_shd);
	digital_input_shadow_cycle(stop_di_shd);
	digital_output_shadow_cycle(stop_lamp_do_shd);
END_IF
END_ACTION

END_PROGRAM

// ---- _Debug/dbg_csp_transfer_main_services_towerlamp.TcPOU

(********************* G.D S.p.A. - Technical Department ***********************************
This program has been generated automatically from Application Designer DE&F
********************************************************************************************)
PROGRAM dbg_csp_transfer_main_services_towerlamp
VAR
  blue_do_shd : digital_output_shadow;
  buzzer_do_shd : digital_output_shadow;
  green_do_shd : digital_output_shadow;
  red_do_shd : digital_output_shadow;
  yellow_do_shd : digital_output_shadow;
END_VAR

_objects_manager();

IF	g_application_status <> APPLICATION_STATUS_RUNNING
THEN
	RETURN;
END_IF

CASE process_get_mode(CONVERSION_this := dbg_root.prc) OF
	MODE_ABSENT,
	MODE_INACTIVE:
		RETURN;
	MODE_TEST:
		RETURN;
END_CASE

ACTION _objects_manager:
IF	objects_initialization()
THEN
	digital_output_shadow_init(
		sim_mode:= SHADOW_SIMULATION_MODE_AUTOMATIC, 
		father:= csp_transfer_main_services_towerlamp.blue_do, 
		process:= dbg_root.prc, 
		CONVERSION_this:= blue_do_shd);

	digital_output_shadow_init(
		sim_mode:= SHADOW_SIMULATION_MODE_AUTOMATIC, 
		father:= csp_transfer_main_services_towerlamp.buzzer_do, 
		process:= dbg_root.prc, 
		CONVERSION_this:= buzzer_do_shd);

	digital_output_shadow_init(
		sim_mode:= SHADOW_SIMULATION_MODE_AUTOMATIC, 
		father:= csp_transfer_main_services_towerlamp.green_do, 
		process:= dbg_root.prc, 
		CONVERSION_this:= green_do_shd);

	digital_output_shadow_init(
		sim_mode:= SHADOW_SIMULATION_MODE_AUTOMATIC, 
		father:= csp_transfer_main_services_towerlamp.red_do, 
		process:= dbg_root.prc, 
		CONVERSION_this:= red_do_shd);

	digital_output_shadow_init(
		sim_mode:= SHADOW_SIMULATION_MODE_AUTOMATIC, 
		father:= csp_transfer_main_services_towerlamp.yellow_do, 
		process:= dbg_root.prc, 
		CONVERSION_this:= yellow_do_shd);

	RETURN;
END_IF

IF	objects_running()
THEN
	digital_output_shadow_cycle(blue_do_shd);
	digital_output_shadow_cycle(buzzer_do_shd);
	digital_output_shadow_cycle(green_do_shd);
	digital_output_shadow_cycle(red_do_shd);
	digital_output_shadow_cycle(yellow_do_shd);
END_IF
END_ACTION

END_PROGRAM

// ---- _Debug/dbg_csp_transfer_upstacker_backstop.TcPOU

(********************* G.D S.p.A. - Technical Department ***********************************
This program has been generated automatically from Application Designer DE&F
********************************************************************************************)
PROGRAM dbg_csp_transfer_upstacker_backstop
VAR
  _sact_shd : digital_actuator_shadow;
  extend_do_shd : digital_output_shadow;
  retracted_di_shd : digital_input_shadow;
END_VAR

_objects_manager();

IF	g_application_status <> APPLICATION_STATUS_RUNNING
THEN
	RETURN;
END_IF

CASE process_get_mode(CONVERSION_this := dbg_root.prc) OF
	MODE_ABSENT,
	MODE_INACTIVE:
		RETURN;
	MODE_TEST:
		RETURN;
END_CASE

ACTION _objects_manager:
IF	objects_initialization()
THEN
	digital_actuator_shadow_init(
		sim_mode:= SHADOW_SIMULATION_MODE_AUTOMATIC, 
		father:= csp_transfer_upstacker_backstop._sact, 
		process:= dbg_root.prc, 
		CONVERSION_this:= _sact_shd);

	digital_output_shadow_init(
		sim_mode:= SHADOW_SIMULATION_MODE_AUTOMATIC, 
		father:= csp_transfer_upstacker_backstop.extend_do, 
		process:= dbg_root.prc, 
		CONVERSION_this:= extend_do_shd);

	digital_input_shadow_init(
		sim_mode:= SHADOW_SIMULATION_MODE_AUTOMATIC, 
		father:= csp_transfer_upstacker_backstop.retracted_di, 
		process:= dbg_root.prc, 
		CONVERSION_this:= retracted_di_shd);

	RETURN;
END_IF

IF	objects_running()
THEN
	digital_actuator_shadow_cycle(_sact_shd);
	digital_output_shadow_cycle(extend_do_shd);
	digital_input_shadow_cycle(retracted_di_shd);
END_IF
END_ACTION

END_PROGRAM

// ---- _Debug/dbg_csp_transfer_upstacker_downstream.TcPOU

(********************* G.D S.p.A. - Technical Department ***********************************
This program has been generated automatically from Application Designer DE&F
********************************************************************************************)
PROGRAM dbg_csp_transfer_upstacker_downstream
VAR
  axis_shd : axis_shadow;
END_VAR

_objects_manager();

IF	g_application_status <> APPLICATION_STATUS_RUNNING
THEN
	RETURN;
END_IF

CASE process_get_mode(CONVERSION_this := dbg_root.prc) OF
	MODE_ABSENT,
	MODE_INACTIVE:
		RETURN;
	MODE_TEST:
		RETURN;
END_CASE

ACTION _objects_manager:
IF	objects_initialization()
THEN
	axis_shadow_init(
		sim_mode:= SHADOW_SIMULATION_MODE_AUTOMATIC, 
		father:= csp_transfer_upstacker_downstream.axis, 
		process:= dbg_root.prc, 
		CONVERSION_this:= axis_shd);

	RETURN;
END_IF

IF	objects_running()
THEN
	axis_shadow_cycle(axis_shd);
END_IF
END_ACTION

END_PROGRAM

// ---- _Debug/dbg_csp_transfer_upstacker_sensors.TcPOU

(********************* G.D S.p.A. - Technical Department ***********************************
This program has been generated automatically from Application Designer DE&F
********************************************************************************************)
PROGRAM dbg_csp_transfer_upstacker_sensors
VAR
  carton_backstop_di_shd : digital_input_shadow;
  prime_di_shd : digital_input_shadow;
END_VAR

_objects_manager();

IF	g_application_status <> APPLICATION_STATUS_RUNNING
THEN
	RETURN;
END_IF

CASE process_get_mode(CONVERSION_this := dbg_root.prc) OF
	MODE_ABSENT,
	MODE_INACTIVE:
		RETURN;
	MODE_TEST:
		RETURN;
END_CASE

ACTION _objects_manager:
IF	objects_initialization()
THEN
	digital_input_shadow_init(
		sim_mode:= SHADOW_SIMULATION_MODE_AUTOMATIC, 
		father:= csp_transfer_upstacker_sensors.carton_backstop_di, 
		process:= dbg_root.prc, 
		CONVERSION_this:= carton_backstop_di_shd);

	digital_input_shadow_init(
		sim_mode:= SHADOW_SIMULATION_MODE_AUTOMATIC, 
		father:= csp_transfer_upstacker_sensors.prime_di, 
		process:= dbg_root.prc, 
		CONVERSION_this:= prime_di_shd);

	RETURN;
END_IF

IF	objects_running()
THEN
	digital_input_shadow_cycle(carton_backstop_di_shd);
	digital_input_shadow_cycle(prime_di_shd);
END_IF
END_ACTION

END_PROGRAM

// ---- _Debug/dbg_csp_transfer_upstacker_upstream.TcPOU

(********************* G.D S.p.A. - Technical Department ***********************************
This program has been generated automatically from Application Designer DE&F
********************************************************************************************)
PROGRAM dbg_csp_transfer_upstacker_upstream
VAR
  axis_shd : axis_shadow;
END_VAR

_objects_manager();

IF	g_application_status <> APPLICATION_STATUS_RUNNING
THEN
	RETURN;
END_IF

CASE process_get_mode(CONVERSION_this := dbg_root.prc) OF
	MODE_ABSENT,
	MODE_INACTIVE:
		RETURN;
	MODE_TEST:
		RETURN;
END_CASE

ACTION _objects_manager:
IF	objects_initialization()
THEN
	axis_shadow_init(
		sim_mode:= SHADOW_SIMULATION_MODE_AUTOMATIC, 
		father:= csp_transfer_upstacker_upstream.axis, 
		process:= dbg_root.prc, 
		CONVERSION_this:= axis_shd);

	RETURN;
END_IF

IF	objects_running()
THEN
	axis_shadow_cycle(axis_shd);
END_IF
END_ACTION

END_PROGRAM

// ---- _Debug/dbg_csp_transfer_upstacker_virtualmaster.TcPOU

(********************* G.D S.p.A. - Technical Department ***********************************
This program has been generated automatically from Application Designer DE&F
********************************************************************************************)
PROGRAM dbg_csp_transfer_upstacker_virtualmaster
VAR
  axis_shd : axis_shadow;
END_VAR

_objects_manager();

IF	g_application_status <> APPLICATION_STATUS_RUNNING
THEN
	RETURN;
END_IF

CASE process_get_mode(CONVERSION_this := dbg_root.prc) OF
	MODE_ABSENT,
	MODE_INACTIVE:
		RETURN;
	MODE_TEST:
		RETURN;
END_CASE

ACTION _objects_manager:
IF	objects_initialization()
THEN
	axis_shadow_init(
		sim_mode:= SHADOW_SIMULATION_MODE_AUTOMATIC, 
		father:= csp_transfer_upstacker_virtualmaster.axis, 
		process:= dbg_root.prc, 
		CONVERSION_this:= axis_shd);

	RETURN;
END_IF

IF	objects_running()
THEN
	axis_shadow_cycle(axis_shd);
END_IF
END_ACTION

END_PROGRAM

// ---- _Debug/dbg_csp_transfer_virtualmaster.TcPOU

(********************* G.D S.p.A. - Technical Department ***********************************
This program has been generated automatically from Application Designer DE&F
********************************************************************************************)
PROGRAM dbg_csp_transfer_virtualmaster
VAR
  axis_shd : axis_shadow;
END_VAR

_objects_manager();

IF	g_application_status <> APPLICATION_STATUS_RUNNING
THEN
	RETURN;
END_IF

CASE process_get_mode(CONVERSION_this := dbg_root.prc) OF
	MODE_ABSENT,
	MODE_INACTIVE:
		RETURN;
	MODE_TEST:
		RETURN;
END_CASE

ACTION _objects_manager:
IF	objects_initialization()
THEN
	axis_shadow_init(
		sim_mode:= SHADOW_SIMULATION_MODE_AUTOMATIC, 
		father:= csp_transfer_virtualmaster.axis, 
		process:= dbg_root.prc, 
		CONVERSION_this:= axis_shd);

	RETURN;
END_IF

IF	objects_running()
THEN
	axis_shadow_cycle(axis_shd);
END_IF
END_ACTION

END_PROGRAM

// ---- _Debug/dbg_quality_checks.TcPOU

(********************* G.D S.p.A. - Technical Department ***********************************
This program has been generated automatically from Application Designer DE&F
********************************************************************************************)
PROGRAM dbg_quality_checks
VAR
  i : DINT;
END_VAR

_objects_manager();

IF	g_application_status <> APPLICATION_STATUS_RUNNING
THEN
	RETURN;
END_IF

CASE process_get_mode(CONVERSION_this := dbg_root.prc) OF
	MODE_ABSENT,
	MODE_INACTIVE:
		RETURN;
	MODE_TEST:
		RETURN;
END_CASE

ACTION _objects_manager:
IF	objects_initialization()
THEN
	RETURN;
END_IF

IF	objects_running()
THEN
	check_section_shadow_cycle(dbg_csp_case_discharge_reject_sensors.reject_trigger_inchoerence_chksect_shd);
	check_section_shadow_cycle(dbg_csp_case_feed_arm_sensors.case_check_chksect_shd);
	check_section_shadow_cycle(dbg_csp_case_feed_arm_sensors.case_check_inchoerence_chksect_shd);
	check_section_shadow_cycle(dbg_csp_case_fc_ls_lower_sensors.flap_chksect_shd);
	check_section_shadow_cycle(dbg_csp_case_fc_ls_upper_sensors.flap_chksect_shd);
	check_section_shadow_cycle(dbg_csp_case_fc_os_lower_sensors.flap_chksect_shd);
	check_section_shadow_cycle(dbg_csp_case_fc_os_upper_sensors.flap_chksect_shd);
	check_section_shadow_cycle(dbg_csp_case_glue_sensors.case_present_ls_di_dchk_shd);
	check_section_shadow_cycle(dbg_csp_case_glue_sensors.case_present_ls_sensor_inchoerence_chksect_shd);
	check_section_shadow_cycle(dbg_csp_case_glue_sensors.case_present_os_di_dchk_shd);
	check_section_shadow_cycle(dbg_csp_case_glue_sensors.case_present_os_sensor_inchoerence_chksect_shd);
	check_section_shadow_cycle(dbg_csp_case_openflap_sensors.open_flap_ls_di_dchk_shd);
	check_section_shadow_cycle(dbg_csp_case_openflap_sensors.open_flap_os_di_dchk_shd);
	;
END_IF
END_ACTION

END_PROGRAM

// ---- _Debug/_Tasks/dbg_highest.TcPOU
PROGRAM dbg_highest
VAR
END_VAR

IF NOT framework_is_local_simulated()
THEN
	RETURN;	
END_IF
dbg_root();
dbg_quality_checks();
dbg_csp_case_closing_ls_horizontal();
dbg_csp_case_closing_ls_lower();
dbg_csp_case_closing_ls_upper();
dbg_csp_case_closing_os_horizontal();
dbg_csp_case_closing_os_lower();
dbg_csp_case_closing_os_upper();
dbg_csp_case_discharge_accu_depth();
dbg_csp_case_discharge_belts_conveyor();
dbg_csp_case_discharge_belts_rotate();
dbg_csp_case_discharge_reject_belt();
dbg_csp_case_discharge_reject_sensors();
dbg_csp_case_discharge_speedbelt_ls();
dbg_csp_case_discharge_speedbelt_os();
dbg_csp_case_feed_arm_elbow();
dbg_csp_case_feed_arm_sensors();
dbg_csp_case_feed_arm_shoulder();
dbg_csp_case_feed_arm_wrist();
dbg_csp_case_feed_kinematic_tilt();
dbg_csp_case_feed_kinematic_x();
dbg_csp_case_feed_kinematic_y();
dbg_csp_case_feed_magazine_accu_lsdepth();
dbg_csp_case_feed_magazine_accu_osdepth();
dbg_csp_case_feed_magazine_level_zone1();
dbg_csp_case_feed_magazine_level_zone2();
dbg_csp_case_feed_magazine_level_zone3();
dbg_csp_case_feed_magazine_level_zonelow();
dbg_csp_case_feed_magazine_level_zonemin();
dbg_csp_case_feed_magazine_ls_belt();
dbg_csp_case_feed_magazine_ls_pusher();
dbg_csp_case_feed_magazine_ls_pushertilt();
dbg_csp_case_feed_magazine_ls_sensors();
dbg_csp_case_feed_magazine_os_belt();
dbg_csp_case_feed_magazine_os_pusher();
dbg_csp_case_feed_magazine_os_pushertilt();
dbg_csp_case_feed_magazine_os_sensors();
dbg_csp_case_feed_reject_belt_lower();
dbg_csp_case_feed_reject_belt_upper();
dbg_csp_case_feed_reject_sensors();
dbg_csp_case_feed_shuttle_accu_depth();
dbg_csp_case_feed_shuttle_horizontal();
dbg_csp_case_feed_shuttle_sensors();
dbg_csp_case_feed_shuttle_sensors_ls();
dbg_csp_case_feed_shuttle_sensors_os();
dbg_csp_case_feed_shuttle_vertical();
dbg_csp_case_fc_ls_lower_follower();
dbg_csp_case_fc_ls_lower_sensors();
dbg_csp_case_fc_ls_lower_spreader();
dbg_csp_case_fc_ls_lower_trailingcloser();
dbg_csp_case_fc_ls_upper_follower();
dbg_csp_case_fc_ls_upper_leadingminorcloser();
dbg_csp_case_fc_ls_upper_sensors();
dbg_csp_case_fc_ls_upper_spreader();
dbg_csp_case_fc_os_lower_follower();
dbg_csp_case_fc_os_lower_sensors();
dbg_csp_case_fc_os_lower_spreader();
dbg_csp_case_fc_os_lower_trailingcloser();
dbg_csp_case_fc_os_upper_follower();
dbg_csp_case_fc_os_upper_sensors();
dbg_csp_case_fc_os_upper_spreader();
dbg_csp_case_glue_hotmelt();
dbg_csp_case_glue_ls_accu_lowerposition();
dbg_csp_case_glue_ls_accu_upperposition();
dbg_csp_case_glue_os_accu_lowerposition();
dbg_csp_case_glue_os_accu_upperposition();
dbg_csp_case_glue_os_accu_width();
dbg_csp_case_glue_virtualmaster();
dbg_csp_case_loader_guide_accu_width();
dbg_csp_case_loader_guide_downstream();
dbg_csp_case_loader_guide_length();
dbg_csp_case_loader_guide_upstream();
dbg_csp_case_main_safety_accuchange();
dbg_csp_case_main_safety_drives_commonconfiguration();
dbg_csp_case_main_safety_drives_ps2000();
dbg_csp_case_main_safety_drives_sd10000();
dbg_csp_case_main_safety_drives_sd10100();
dbg_csp_case_main_safety_drives_sd10200();
dbg_csp_case_main_safety_drives_sd10300();
dbg_csp_case_main_safety_drives_sd10400();
dbg_csp_case_main_safety_drives_sd11000();
dbg_csp_case_main_safety_drives_sd12000();
dbg_csp_case_main_safety_drives_sd15000();
dbg_csp_case_main_safety_drives_sd2100();
dbg_csp_case_main_safety_drives_sd2200();
dbg_csp_case_main_safety_drives_sd2300();
dbg_csp_case_main_safety_drives_sd2400();
dbg_csp_case_main_safety_drives_sd2500();
dbg_csp_case_main_safety_drives_sd26000();
dbg_csp_case_main_safety_drives_sd26100();
dbg_csp_case_main_safety_drives_sd8000();
dbg_csp_case_main_safety_drives_sd8100();
dbg_csp_case_main_safety_drives_sd8200();
dbg_csp_case_main_safety_drives_sd8300();
dbg_csp_case_main_safety_drives_sd8400();
dbg_csp_case_main_safety_drives_sd8500();
dbg_csp_case_main_safety_drives_sd8600();
dbg_csp_case_main_safety_emergency();
dbg_csp_case_main_safety_guards();
dbg_csp_case_openflap_sensors();
dbg_csp_case_tr_accu_depth();
dbg_csp_case_tr_accu_ls_width();
dbg_csp_case_tr_accu_os_width();
dbg_csp_case_tr_squaring_ls_leading();
dbg_csp_case_tr_squaring_ls_trailing();
dbg_csp_case_tr_squaring_os_leading();
dbg_csp_case_tr_squaring_os_trailing();
dbg_csp_case_transport_accu_depth();
dbg_csp_case_transport_ls_leading();
dbg_csp_case_transport_ls_trailing();
dbg_csp_case_transport_os_leading();
dbg_csp_case_transport_os_minorplow();
dbg_csp_case_transport_os_trailing();
dbg_csp_case_transport_virtualmaster();
dbg_csp_main_motorization_virtualmanager();
dbg_csp_transfer_accumulator_accu_convdepth();
dbg_csp_transfer_accumulator_accu_depth();
dbg_csp_transfer_accumulator_accu_topraillength();
dbg_csp_transfer_accumulator_accu_toprailwidth();
dbg_csp_transfer_accumulator_belt();
dbg_csp_transfer_accumulator_finger_ls();
dbg_csp_transfer_accumulator_finger_os();
dbg_csp_transfer_accumulator_lift();
dbg_csp_transfer_accumulator_virtualmaster();
dbg_csp_transfer_infeed();

END_PROGRAM

// ---- _Debug/_Tasks/dbg_low.TcPOU
PROGRAM dbg_low
VAR
END_VAR

IF NOT framework_is_local_simulated()
THEN
	RETURN;	
END_IF
dbg_csp_main_jogmanager();
dbg_csp_transfer_main_safety_drives_commonconfiguration();
dbg_csp_transfer_infeed_accu_depth();
dbg_csp_transfer_infeed_accu_waterfalladjust();
dbg_csp_transfer_infeed_accumulation_belt();
dbg_csp_transfer_infeed_accumulation_level_low();
dbg_csp_transfer_infeed_accumulation_level_max();
dbg_csp_transfer_infeed_accumulation_level_min();
dbg_csp_transfer_infeed_accumulation_level_normal();
dbg_csp_transfer_infeed_metering_belt();
dbg_csp_transfer_infeed_metering_jam();
dbg_csp_transfer_infeed_waterfall_belt();
dbg_csp_transfer_main_safety_accuchange();
dbg_csp_transfer_main_safety_drives_ps41020();
dbg_csp_transfer_main_safety_drives_sd41100();
dbg_csp_transfer_main_safety_drives_sd41200();
dbg_csp_transfer_main_safety_drives_sd41300();
dbg_csp_transfer_main_safety_drives_sd41400();
dbg_csp_transfer_main_safety_drives_sd41500();
dbg_csp_transfer_main_safety_drives_sd41600();
dbg_csp_transfer_main_safety_drives_sd41700();
dbg_csp_transfer_main_safety_emergency();
dbg_csp_transfer_main_safety_guards();
dbg_csp_transfer_main_safety_token();

END_PROGRAM

// ---- _Debug/_Tasks/dbg_lowest.TcPOU
PROGRAM dbg_lowest
VAR
END_VAR

IF NOT framework_is_local_simulated()
THEN
	RETURN;	
END_IF

END_PROGRAM

// ---- _Debug/_Tasks/dbg_normal.TcPOU
PROGRAM dbg_normal
VAR
END_VAR

IF NOT framework_is_local_simulated()
THEN
	RETURN;	
END_IF
dbg_csp_case_feed_virtualmaster();
dbg_csp_case_flapcontrol_backstop();
dbg_csp_case_glue_sensors();
dbg_csp_case_loader_pusher();
dbg_csp_case_loader_virtualmaster();
dbg_csp_case_main_services();
dbg_csp_case_main_services_breakers();
dbg_csp_case_main_services_pushbuttons();
dbg_csp_case_transport_tensioner();
dbg_csp_case_virtualmaster();
dbg_csp_main_services();
dbg_csp_transfer_crosspusher_follower();
dbg_csp_transfer_crosspusher_horizontal();
dbg_csp_transfer_crosspusher_reject();
dbg_csp_transfer_crosspusher_sensors();
dbg_csp_transfer_crosspusher_vertical();
dbg_csp_transfer_crosspusher_virtualmaster();
dbg_csp_transfer_infeed_clamp();
dbg_csp_transfer_infeed_reject_highload();
dbg_csp_transfer_infeed_reject_pusher();
dbg_csp_transfer_infeed_reject_virtualmaster();
dbg_csp_transfer_main_services();
dbg_csp_transfer_main_services_breakers();
dbg_csp_transfer_main_services_pushbuttons();
dbg_csp_transfer_main_services_towerlamp();
dbg_csp_transfer_upstacker_backstop();
dbg_csp_transfer_upstacker_downstream();
dbg_csp_transfer_upstacker_sensors();
dbg_csp_transfer_upstacker_upstream();
dbg_csp_transfer_upstacker_virtualmaster();
dbg_csp_transfer_virtualmaster();

END_PROGRAM

